LIN {X 0,Y 303.853,Z 837.936,A -85,B 0,C 180,E1 -16106.02,E2 -16106.02} C_VEL
LIN {X 0,Y 303.612,Z 839.547,A -85,B 0,C 180,E1 -16108.673,E2 -16108.673} C_VEL
LIN {X 0,Y 303.609,Z 839.78,A -85,B 0,C 180,E1 -16109.999,E2 -16109.999} C_VEL
LIN {X 0,Y 303.611,Z 839.586,A -85,B 0,C 180,E1 -16111.325,E2 -16111.325} C_VEL
LIN {X 0,Y 303.847,Z 838.029,A -85,B 0,C 180,E1 -16113.978,E2 -16113.978} C_VEL
LIN {X 0,Y 303.974,Z 836.663,A -85,B 0,C 180,E1 -16115.305,E2 -16115.305} C_VEL
LIN {X 0,Y 304.327,Z 833.787,A -85,B 0,C 180,E1 -16117.296,E2 -16117.296} C_VEL
LIN {X 0,Y 304.835,Z 829.878,A -85,B 0,C 180,E1 -16119.286,E2 -16119.286} C_VEL
LIN {X 0,Y 305.628,Z 824.814,A -85,B 0,C 180,E1 -16121.27,E2 -16121.27} C_VEL
LIN {X 0,Y 306.668,Z 818.43,A -85,B 0,C 180,E1 -16123.247,E2 -16123.247} C_VEL
LIN {X 0,Y 308.069,Z 810.481,A -85,B 0,C 180,E1 -16125.208,E2 -16125.208} C_VEL
LIN {X 0,Y 309.461,Z 802.349,A -85,B 0,C 180,E1 -16126.83,E2 -16126.83} C_VEL
LIN {X 0,Y 310.862,Z 792.359,A -85,B 0,C 180,E1 -16128.451,E2 -16128.451} C_VEL
LIN {X 0,Y 312.33,Z 781.127,A -85,B 0,C 180,E1 -16129.896,E2 -16129.896} C_VEL
LIN {X 0,Y 313.671,Z 770.081,A -85,B 0,C 180,E1 -16131.006,E2 -16131.006} C_VEL
LIN {X 0,Y 314.929,Z 757.587,A -85,B 0,C 180,E1 -16131.948,E2 -16131.948} C_VEL
LIN {X 0,Y 315.711,Z 745.352,A -85,B 0,C 180,E1 -16132.623,E2 -16132.623} C_VEL
LIN {X 0,Y 316.307,Z 733.163,A -85,B 0,C 180,E1 -16133.053,E2 -16133.053} C_VEL
LIN {X 0,Y 318.131,Z 657.232,A -85,B 0,C 180,E1 -16134.766,E2 -16134.766} C_VEL
LIN {X 0,Y 314.244,Z 634.232,A -85,B 0,C 180,E1 -16135.666,E2 -16135.666} C_VEL
LIN {X 0,Y 312.534,Z 625.542,A -85,B 0,C 180,E1 -16136.042,E2 -16136.042} C_VEL
LIN {X 0,Y 313.811,Z 610.673,A -85,B 0,C 180,E1 -16138.901,E2 -16138.901} C_VEL
LIN {X 0,Y 314.735,Z 599.426,A -85,B 0,C 180,E1 -16141.163,E2 -16141.163} C_VEL
LIN {X 0,Y 312.386,Z 587.67,A -85,B 0,C 180,E1 -16143.984,E2 -16143.984} C_VEL
LIN {X 0,Y 309.121,Z 574.667,A -85,B 0,C 180,E1 -16147.274,E2 -16147.274} C_VEL
LIN {X 0,Y 308.68,Z 573.104,A -85,B 0,C 180,E1 -16147.688,E2 -16147.688} C_VEL
LIN {X 0,Y 307.449,Z 571.218,A -85,B 0,C 180,E1 -16148.289,E2 -16148.289} C_VEL
LIN {X 0,Y 303.889,Z 568.949,A -85,B 0,C 180,E1 -16149.268,E2 -16149.268} C_VEL
LIN {X 0,Y 300.215,Z 566.767,A -85,B 0,C 180,E1 -16150.27,E2 -16150.27} C_VEL
LIN {X 0,Y 298.831,Z 564.916,A -85,B 0,C 180,E1 -16150.899,E2 -16150.899} C_VEL
LIN {X 0,Y 298.391,Z 563.319,A -85,B 0,C 180,E1 -16151.371,E2 -16151.371} C_VEL
LIN {X 0,Y 298.431,Z 563.292,A -85,B 0,C 180,E1 -16154.237,E2 -16154.237} C_VEL
LIN {X 0,Y 307.008,Z 587.38,A -85,B 0,C 180,E1 -16155.516,E2 -16155.516} C_VEL
LIN {X 0,Y 305.715,Z 636.753,A -85,B 0,C 180,E1 -16156.941,E2 -16156.941} C_VEL
LIN {X 0,Y 305.575,Z 650.861,A -85,B 0,C 180,E1 -16157.466,E2 -16157.466} C_VEL
LIN {X 0,Y 305.157,Z 664.019,A -85,B 0,C 180,E1 -16158.217,E2 -16158.217} C_VEL
LIN {X 0,Y 304.525,Z 676.406,A -85,B 0,C 180,E1 -16159.176,E2 -16159.176} C_VEL
LIN {X 0,Y 303.715,Z 689.144,A -85,B 0,C 180,E1 -16160.479,E2 -16160.479} C_VEL
LIN {X 0,Y 302.952,Z 699.146,A -85,B 0,C 180,E1 -16161.754,E2 -16161.754} C_VEL
LIN {X 0,Y 302.031,Z 709.642,A -85,B 0,C 180,E1 -16163.396,E2 -16163.396} C_VEL
LIN {X 0,Y 301.174,Z 718.74,A -85,B 0,C 180,E1 -16165.152,E2 -16165.152} C_VEL
LIN {X 0,Y 300.4,Z 726.936,A -85,B 0,C 180,E1 -16167.087,E2 -16167.087} C_VEL
LIN {X 0,Y 299.749,Z 733.339,A -85,B 0,C 180,E1 -16168.948,E2 -16168.948} C_VEL
LIN {X 0,Y 299.288,Z 739.52,A -85,B 0,C 180,E1 -16171.224,E2 -16171.224} C_VEL
LIN {X 0,Y 298.93,Z 744.17,A -85,B 0,C 180,E1 -16173.468,E2 -16173.468} C_VEL
LIN {X 0,Y 298.784,Z 746.542,A -85,B 0,C 180,E1 -16174.951,E2 -16174.951} C_VEL
LIN {X 0,Y 298.8,Z 748.429,A -85,B 0,C 180,E1 -16176.531,E2 -16176.531} C_VEL
LIN {X 0,Y 298.875,Z 749.634,A -85,B 0,C 180,E1 -16177.899,E2 -16177.899} C_VEL
LIN {X 0,Y 299.187,Z 750.596,A -85,B 0,C 180,E1 -16179.981,E2 -16179.981} C_VEL
LIN {X 0,Y 299.717,Z 750.5,A -85,B 0,C 180,E1 -16182.252,E2 -16182.252} C_VEL
LIN {X 0,Y 300.208,Z 749.793,A -85,B 0,C 180,E1 -16183.698,E2 -16183.698} C_VEL
LIN {X 0,Y 300.767,Z 748.669,A -85,B 0,C 180,E1 -16185.106,E2 -16185.106} C_VEL
LIN {X 0,Y 301.416,Z 747.031,A -85,B 0,C 180,E1 -16186.516,E2 -16186.516} C_VEL
LIN {X 0,Y 302.579,Z 743.644,A -85,B 0,C 180,E1 -16188.613,E2 -16188.613} C_VEL
LIN {X 0,Y 304.012,Z 739.036,A -85,B 0,C 180,E1 -16190.687,E2 -16190.687} C_VEL
LIN {X 0,Y 305.628,Z 733.047,A -85,B 0,C 180,E1 -16192.756,E2 -16192.756} C_VEL
LIN {X 0,Y 307.449,Z 725.584,A -85,B 0,C 180,E1 -16194.754,E2 -16194.754} C_VEL
LIN {X 0,Y 309.25,Z 717.437,A -85,B 0,C 180,E1 -16196.5,E2 -16196.5} C_VEL
LIN {X 0,Y 310.935,Z 708.306,A -85,B 0,C 180,E1 -16198.099,E2 -16198.099} C_VEL
LIN {X 0,Y 312.621,Z 698.14,A -85,B 0,C 180,E1 -16199.517,E2 -16199.517} C_VEL
LIN {X 0,Y 314.131,Z 686.583,A -85,B 0,C 180,E1 -16200.801,E2 -16200.801} C_VEL
LIN {X 0,Y 315.358,Z 674.542,A -85,B 0,C 180,E1 -16201.836,E2 -16201.836} C_VEL
LIN {X 0,Y 316.231,Z 660.72,A -85,B 0,C 180,E1 -16202.723,E2 -16202.723} C_VEL
LIN {X 0,Y 316.632,Z 647.103,A -85,B 0,C 180,E1 -16203.316,E2 -16203.316} C_VEL
LIN {X 0,Y 317.899,Z 617.446,A -85,B 0,C 180,E1 -16204.302,E2 -16204.302} C_VEL
LIN {X 0,Y 318.949,Z 597.845,A -85,B 0,C 180,E1 -16204.935,E2 -16204.935} C_VEL
LIN {X 0,Y 314.572,Z 589.417,A -85,B 0,C 180,E1 -16205.965,E2 -16205.965} C_VEL
LIN {X 0,Y 306.906,Z 576.235,A -85,B 0,C 180,E1 -16207.897,E2 -16207.897} C_VEL
LIN {X 0,Y 304.292,Z 572.293,A -85,B 0,C 180,E1 -16208.591,E2 -16208.591} C_VEL
LIN {X 0,Y 302.125,Z 569.115,A -85,B 0,C 180,E1 -16209.179,E2 -16209.179} C_VEL
LIN {X 0,Y 301.351,Z 567.986,A -85,B 0,C 180,E1 -16209.396,E2 -16209.396} C_VEL
LIN {X 0,Y 299.391,Z 565.714,A -85,B 0,C 180,E1 -16209.943,E2 -16209.943} C_VEL
LIN {X 0,Y 298.616,Z 563.282,A -85,B 0,C 180,E1 -16210.274,E2 -16210.274} C_VEL
LIN {X 0,Y 298.584,Z 563.287,A -85,B 0,C 180,E1 -16215.006,E2 -16215.006} C_VEL
LIN {X 0,Y 298.53,Z 563.298,A -85,B 0,C 180,E1 -16219.244,E2 -16219.244} C_VEL
LIN {X 0,Y 298.449,Z 563.309,A -85,B 0,C 180,E1 -16223.598,E2 -16223.598} C_VEL
LIN {X 0,Y 298.481,Z 563.304,A -85,B 0,C 180,E1 -16226.575,E2 -16226.575} C_VEL
LIN {X 0,Y 298.413,Z 563.313,A -85,B 0,C 180,E1 -16229.642,E2 -16229.642} C_VEL
LIN {X 0,Y 298.388,Z 563.317,A -85,B 0,C 180,E1 -16232.801,E2 -16232.801} C_VEL
LIN {X 0,Y 298.459,Z 563.304,A -85,B 0,C 180,E1 -16236.814,E2 -16236.814} C_VEL
LIN {X 0,Y 298.45,Z 563.309,A -85,B 0,C 180,E1 -16241.104,E2 -16241.104} C_VEL
LIN {X 0,Y 298.471,Z 563.304,A -85,B 0,C 180,E1 -16242.607,E2 -16242.607} C_VEL
LIN {X 0,Y 300.836,Z 570.374,A -85,B 0,C 180,E1 -16246.403,E2 -16246.403} C_VEL
LIN {X 0,Y 303.269,Z 578.289,A -85,B 0,C 180,E1 -16249.885,E2 -16249.885} C_VEL
LIN {X 0,Y 305.728,Z 587.467,A -85,B 0,C 180,E1 -16253.298,E2 -16253.298} C_VEL
LIN {X 0,Y 307.819,Z 597.274,A -85,B 0,C 180,E1 -16256.458,E2 -16256.458} C_VEL
LIN {X 0,Y 308.48,Z 601.915,A -85,B 0,C 180,E1 -16257.793,E2 -16257.793} C_VEL
LIN {X 0,Y 307.38,Z 607.823,A -85,B 0,C 180,E1 -16259.17,E2 -16259.17} C_VEL
LIN {X 0,Y 311.06,Z 628.758,A -85,B 0,C 180,E1 -16260.676,E2 -16260.676} C_VEL
LIN {X 0,Y 313.364,Z 646.451,A -85,B 0,C 180,E1 -16261.741,E2 -16261.741} C_VEL
LIN {X 0,Y 314.792,Z 663.123,A -85,B 0,C 180,E1 -16262.607,E2 -16262.607} C_VEL
LIN {X 0,Y 315.561,Z 682.154,A -85,B 0,C 180,E1 -16263.427,E2 -16263.427} C_VEL
LIN {X 0,Y 313.252,Z 724.371,A -85,B 0,C 180,E1 -16264.743,E2 -16264.743} C_VEL
LIN {X 0,Y 311.907,Z 737.532,A -85,B 0,C 180,E1 -16265.366,E2 -16265.366} C_VEL
LIN {X 0,Y 310.311,Z 749.164,A -85,B 0,C 180,E1 -16266.121,E2 -16266.121} C_VEL
LIN {X 0,Y 308.409,Z 760.554,A -85,B 0,C 180,E1 -16267.032,E2 -16267.032} C_VEL
LIN {X 0,Y 307.364,Z 773.902,A -85,B 0,C 180,E1 -16267.748,E2 -16267.748} C_VEL
LIN {X 0,Y 306.138,Z 785.541,A -85,B 0,C 180,E1 -16268.628,E2 -16268.628} C_VEL
LIN {X 0,Y 304.724,Z 796.825,A -85,B 0,C 180,E1 -16269.762,E2 -16269.762} C_VEL
LIN {X 0,Y 303.078,Z 808.262,A -85,B 0,C 180,E1 -16271.233,E2 -16271.233} C_VEL
LIN {X 0,Y 301.636,Z 817.897,A -85,B 0,C 180,E1 -16272.801,E2 -16272.801} C_VEL
LIN {X 0,Y 300.132,Z 827.345,A -85,B 0,C 180,E1 -16274.727,E2 -16274.727} C_VEL
LIN {X 0,Y 298.789,Z 835.261,A -85,B 0,C 180,E1 -16276.743,E2 -16276.743} C_VEL
LIN {X 0,Y 297.966,Z 840.605,A -85,B 0,C 180,E1 -16278.436,E2 -16278.436} C_VEL
LIN {X 0,Y 297.288,Z 845.825,A -85,B 0,C 180,E1 -16280.476,E2 -16280.476} C_VEL
LIN {X 0,Y 296.856,Z 849.862,A -85,B 0,C 180,E1 -16282.519,E2 -16282.519} C_VEL
LIN {X 0,Y 296.64,Z 852.837,A -85,B 0,C 180,E1 -16284.563,E2 -16284.563} C_VEL
LIN {X 0,Y 296.633,Z 854.265,A -85,B 0,C 180,E1 -16285.925,E2 -16285.925} C_VEL
LIN {X 0,Y 296.613,Z 855.272,A -85,B 0,C 180,E1 -16287.285,E2 -16287.285} C_VEL
LIN {X 0,Y 296.59,Z 855.887,A -85,B 0,C 180,E1 -16288.643,E2 -16288.643} C_VEL
LIN {X 0,Y 296.637,Z 856.105,A -85,B 0,C 180,E1 -16290.001,E2 -16290.001} C_VEL
LIN {X 0,Y 296.608,Z 855.258,A -85,B 0,C 180,E1 -16292.717,E2 -16292.717} C_VEL
LIN {X 0,Y 296.625,Z 854.245,A -85,B 0,C 180,E1 -16294.077,E2 -16294.077} C_VEL
LIN {X 0,Y 296.667,Z 852.404,A -85,B 0,C 180,E1 -16295.745,E2 -16295.745} C_VEL
LIN {X 0,Y 296.984,Z 848.58,A -85,B 0,C 180,E1 -16298.164,E2 -16298.164} C_VEL
LIN {X 0,Y 297.462,Z 844.157,A -85,B 0,C 180,E1 -16300.208,E2 -16300.208} C_VEL
LIN {X 0,Y 298.393,Z 837.421,A -85,B 0,C 180,E1 -16302.585,E2 -16302.585} C_VEL
LIN {X 0,Y 299.642,Z 830.074,A -85,B 0,C 180,E1 -16304.605,E2 -16304.605} C_VEL
LIN {X 0,Y 301.09,Z 821.3,A -85,B 0,C 180,E1 -16306.539,E2 -16306.539} C_VEL
LIN {X 0,Y 302.472,Z 811.371,A -85,B 0,C 180,E1 -16308.282,E2 -16308.282} C_VEL
LIN {X 0,Y 304.14,Z 800.779,A -85,B 0,C 180,E1 -16309.753,E2 -16309.753} C_VEL
LIN {X 0,Y 305.54,Z 790.516,A -85,B 0,C 180,E1 -16310.888,E2 -16310.888} C_VEL
LIN {X 0,Y 306.863,Z 778.19,A -85,B 0,C 180,E1 -16311.939,E2 -16311.939} C_VEL
LIN {X 0,Y 308.027,Z 765.239,A -85,B 0,C 180,E1 -16312.735,E2 -16312.735} C_VEL
LIN {X 0,Y 308.875,Z 752.279,A -85,B 0,C 180,E1 -16313.244,E2 -16313.244} C_VEL
LIN {X 0,Y 310.541,Z 681.414,A -85,B 0,C 180,E1 -16314.888,E2 -16314.888} C_VEL
LIN {X 0,Y 307.31,Z 650.705,A -85,B 0,C 180,E1 -16315.941,E2 -16315.941} C_VEL
LIN {X 0,Y 305.214,Z 635.339,A -85,B 0,C 180,E1 -16316.537,E2 -16316.537} C_VEL
LIN {X 0,Y 303.765,Z 612.724,A -85,B 0,C 180,E1 -16318.456,E2 -16318.456} C_VEL
LIN {X 0,Y 303.073,Z 604.261,A -85,B 0,C 180,E1 -16319.143,E2 -16319.143} C_VEL
LIN {X 0,Y 304.618,Z 592.104,A -85,B 0,C 180,E1 -16322.05,E2 -16322.05} C_VEL
LIN {X 0,Y 302.355,Z 581.022,A -85,B 0,C 180,E1 -16324.963,E2 -16324.963} C_VEL
LIN {X 0,Y 299.36,Z 567.37,A -85,B 0,C 180,E1 -16328.733,E2 -16328.733} C_VEL
LIN {X 0,Y 298.435,Z 563.311,A -85,B 0,C 180,E1 -16329.921,E2 -16329.921} C_VEL
LIN {X 0,Y 298.401,Z 563.308,A -85,B 0,C 180,E1 -16333.104,E2 -16333.104} C_VEL
LIN {X 0,Y 298.405,Z 563.311,A -85,B 0,C 180,E1 -16336.921,E2 -16336.921} C_VEL
LIN {X 0,Y 298.401,Z 563.317,A -85,B 0,C 180,E1 -16341.008,E2 -16341.008} C_VEL
LIN {X 0,Y 298.42,Z 563.299,A -85,B 0,C 180,E1 -16343.93,E2 -16343.93} C_VEL
LIN {X 0,Y 298.397,Z 563.302,A -85,B 0,C 180,E1 -16347.984,E2 -16347.984} C_VEL
LIN {X 0,Y 298.465,Z 563.307,A -85,B 0,C 180,E1 -16351.904,E2 -16351.904} C_VEL
LIN {X 0,Y 298.485,Z 563.284,A -85,B 0,C 180,E1 -16354.924,E2 -16354.924} C_VEL
LIN {X 0,Y 298.441,Z 563.309,A -85,B 0,C 180,E1 -16359.315,E2 -16359.315} C_VEL
LIN {X 0,Y 298.539,Z 563.271,A -85,B 0,C 180,E1 -16362.179,E2 -16362.179} C_VEL
LIN {X 0,Y 298.595,Z 563.287,A -85,B 0,C 180,E1 -16364.995,E2 -16364.995} C_VEL
LIN {X 0,Y 298.593,Z 563.266,A -85,B 0,C 180,E1 -16369.147,E2 -16369.147} C_VEL
LIN {X 0,Y 298.743,Z 563.264,A -85,B 0,C 180,E1 -16371.886,E2 -16371.886} C_VEL
LIN {X 0,Y 298.659,Z 563.279,A -85,B 0,C 180,E1 -16374.599,E2 -16374.599} C_VEL
LIN {X 0,Y 298.923,Z 563.232,A -85,B 0,C 180,E1 -16378.653,E2 -16378.653} C_VEL
LIN {X 0,Y 298.925,Z 563.25,A -85,B 0,C 180,E1 -16381.347,E2 -16381.347} C_VEL
LIN {X 0,Y 298.794,Z 563.254,A -85,B 0,C 180,E1 -16386.754,E2 -16386.754} C_VEL
LIN {X 0,Y 298.682,Z 563.281,A -85,B 0,C 180,E1 -16389.48,E2 -16389.48} C_VEL
LIN {X 0,Y 298.553,Z 563.278,A -85,B 0,C 180,E1 -16393.615,E2 -16393.615} C_VEL
LIN {X 0,Y 298.551,Z 563.295,A -85,B 0,C 180,E1 -16396.409,E2 -16396.409} C_VEL
LIN {X 0,Y 298.513,Z 563.28,A -85,B 0,C 180,E1 -16399.654,E2 -16399.654} C_VEL
LIN {X 0,Y 298.46,Z 563.303,A -85,B 0,C 180,E1 -16403.598,E2 -16403.598} C_VEL
LIN {X 0,Y 298.487,Z 563.294,A -85,B 0,C 180,E1 -16406.575,E2 -16406.575} C_VEL
LIN {X 0,Y 298.419,Z 563.305,A -85,B 0,C 180,E1 -16409.641,E2 -16409.641} C_VEL
LIN {X 0,Y 298.397,Z 563.318,A -85,B 0,C 180,E1 -16412.8,E2 -16412.8} C_VEL
LIN {X 0,Y 298.466,Z 563.307,A -85,B 0,C 180,E1 -16416.812,E2 -16416.812} C_VEL
LIN {X 0,Y 298.39,Z 563.319,A -85,B 0,C 180,E1 -16421.088,E2 -16421.088} C_VEL
LIN {X 0,Y 298.401,Z 563.307,A -85,B 0,C 180,E1 -16423.103,E2 -16423.103} C_VEL
LIN {X 0,Y 298.406,Z 563.29,A -85,B 0,C 180,E1 -16426.921,E2 -16426.921} C_VEL
LIN {X 0,Y 298.43,Z 563.37,A -85,B 0,C 180,E1 -16430.401,E2 -16430.401} C_VEL
LIN {X 0,Y 302.152,Z 575.058,A -85,B 0,C 180,E1 -16433.365,E2 -16433.365} C_VEL
LIN {X 0,Y 305.463,Z 587.296,A -85,B 0,C 180,E1 -16436.257,E2 -16436.257} C_VEL
LIN {X 0,Y 308.042,Z 598.396,A -85,B 0,C 180,E1 -16438.732,E2 -16438.732} C_VEL
LIN {X 0,Y 308.779,Z 602.347,A -85,B 0,C 180,E1 -16439.574,E2 -16439.574} C_VEL
LIN {X 0,Y 307.17,Z 620.347,A -85,B 0,C 180,E1 -16442.767,E2 -16442.767} C_VEL
LIN {X 0,Y 306.845,Z 624.941,A -85,B 0,C 180,E1 -16443.537,E2 -16443.537} C_VEL
LIN {X 0,Y 311.493,Z 653.75,A -85,B 0,C 180,E1 -16444.695,E2 -16444.695} C_VEL
LIN {X 0,Y 311.626,Z 659.554,A -85,B 0,C 180,E1 -16444.852,E2 -16444.852} C_VEL
LIN {X 0,Y 309.66,Z 736.424,A -85,B 0,C 180,E1 -16446.642,E2 -16446.642} C_VEL
LIN {X 0,Y 308.963,Z 749.181,A -85,B 0,C 180,E1 -16447.162,E2 -16447.162} C_VEL
LIN {X 0,Y 307.876,Z 762.003,A -85,B 0,C 180,E1 -16447.961,E2 -16447.961} C_VEL
LIN {X 0,Y 306.553,Z 774.243,A -85,B 0,C 180,E1 -16449.008,E2 -16449.008} C_VEL
LIN {X 0,Y 305.168,Z 784.527,A -85,B 0,C 180,E1 -16450.141,E2 -16450.141} C_VEL
LIN {X 0,Y 303.816,Z 794.443,A -85,B 0,C 180,E1 -16451.52,E2 -16451.52} C_VEL
LIN {X 0,Y 302.426,Z 803.706,A -85,B 0,C 180,E1 -16453.112,E2 -16453.112} C_VEL
LIN {X 0,Y 300.731,Z 813.082,A -85,B 0,C 180,E1 -16455.103,E2 -16455.103} C_VEL
LIN {X 0,Y 299.443,Z 820.531,A -85,B 0,C 180,E1 -16457.116,E2 -16457.116} C_VEL
LIN {X 0,Y 298.397,Z 826.513,A -85,B 0,C 180,E1 -16459.138,E2 -16459.138} C_VEL
LIN {X 0,Y 297.631,Z 831.239,A -85,B 0,C 180,E1 -16461.17,E2 -16461.17} C_VEL
LIN {X 0,Y 297.107,Z 835.247,A -85,B 0,C 180,E1 -16463.467,E2 -16463.467} C_VEL
LIN {X 0,Y 296.769,Z 838.129,A -85,B 0,C 180,E1 -16465.925,E2 -16465.925} C_VEL
LIN {X 0,Y 296.531,Z 839.74,A -85,B 0,C 180,E1 -16468.641,E2 -16468.641} C_VEL
LIN {X 0,Y 296.525,Z 839.973,A -85,B 0,C 180,E1 -16469.999,E2 -16469.999} C_VEL
LIN {X 0,Y 296.53,Z 839.779,A -85,B 0,C 180,E1 -16471.357,E2 -16471.357} C_VEL
LIN {X 0,Y 296.764,Z 838.222,A -85,B 0,C 180,E1 -16474.073,E2 -16474.073} C_VEL
LIN {X 0,Y 297.076,Z 835.498,A -85,B 0,C 180,E1 -16476.48,E2 -16476.48} C_VEL
LIN {X 0,Y 297.606,Z 831.47,A -85,B 0,C 180,E1 -16478.828,E2 -16478.828} C_VEL
LIN {X 0,Y 298.362,Z 826.807,A -85,B 0,C 180,E1 -16480.861,E2 -16480.861} C_VEL
LIN {X 0,Y 299.394,Z 820.897,A -85,B 0,C 180,E1 -16482.884,E2 -16482.884} C_VEL
LIN {X 0,Y 300.668,Z 813.536,A -85,B 0,C 180,E1 -16484.898,E2 -16484.898} C_VEL
LIN {X 0,Y 302.078,Z 805.993,A -85,B 0,C 180,E1 -16486.558,E2 -16486.558} C_VEL
LIN {X 0,Y 303.654,Z 795.708,A -85,B 0,C 180,E1 -16488.388,E2 -16488.388} C_VEL
LIN {X 0,Y 305.131,Z 785.367,A -85,B 0,C 180,E1 -16489.859,E2 -16489.859} C_VEL
LIN {X 0,Y 306.481,Z 775.33,A -85,B 0,C 180,E1 -16490.994,E2 -16490.994} C_VEL
LIN {X 0,Y 307.813,Z 763.399,A -85,B 0,C 180,E1 -16492.041,E2 -16492.041} C_VEL
LIN {X 0,Y 308.86,Z 750.384,A -85,B 0,C 180,E1 -16492.888,E2 -16492.888} C_VEL
LIN {X 0,Y 309.637,Z 737.22,A -85,B 0,C 180,E1 -16493.446,E2 -16493.446} C_VEL
LIN {X 0,Y 311.73,Z 659.363,A -85,B 0,C 180,E1 -16495.257,E2 -16495.257} C_VEL
LIN {X 0,Y 309.107,Z 642.217,A -85,B 0,C 180,E1 -16495.923,E2 -16495.923} C_VEL
LIN {X 0,Y 305.998,Z 625.586,A -85,B 0,C 180,E1 -16496.668,E2 -16496.668} C_VEL
LIN {X 0,Y 307.473,Z 608.89,A -85,B 0,C 180,E1 -16499.915,E2 -16499.915} C_VEL
LIN {X 0,Y 308.081,Z 602.29,A -85,B 0,C 180,E1 -16501.262,E2 -16501.262} C_VEL
LIN {X 0,Y 306.536,Z 593.373,A -85,B 0,C 180,E1 -16503.382,E2 -16503.382} C_VEL
LIN {X 0,Y 303.751,Z 581.527,A -85,B 0,C 180,E1 -16506.401,E2 -16506.401} C_VEL
LIN {X 0,Y 300.486,Z 569.988,A -85,B 0,C 180,E1 -16509.481,E2 -16509.481} C_VEL
LIN {X 0,Y 298.831,Z 564.916,A -85,B 0,C 180,E1 -16510.899,E2 -16510.899} C_VEL
LIN {X 0,Y 298.207,Z 564.181,A -85,B 0,C 180,E1 -16511.434,E2 -16511.434} C_VEL
LIN {X 0,Y 297.663,Z 564.724,A -85,B 0,C 180,E1 -16512.005,E2 -16512.005} C_VEL
LIN {X 0,Y 297.105,Z 566.972,A -85,B 0,C 180,E1 -16512.788,E2 -16512.788} C_VEL
LIN {X 0,Y 296.868,Z 571.244,A -85,B 0,C 180,E1 -16513.605,E2 -16513.605} C_VEL
LIN {X 0,Y 297.126,Z 576.758,A -85,B 0,C 180,E1 -16514.323,E2 -16514.323} C_VEL
LIN {X 0,Y 298.201,Z 582.694,A -85,B 0,C 180,E1 -16514.845,E2 -16514.845} C_VEL
LIN {X 0,Y 298.815,Z 584.718,A -85,B 0,C 180,E1 -16514.965,E2 -16514.965} C_VEL
LIN {X 0,Y 300.204,Z 588.9,A -85,B 0,C 180,E1 -16515.177,E2 -16515.177} C_VEL
LIN {X 0,Y 298.863,Z 635.716,A -85,B 0,C 180,E1 -16516.565,E2 -16516.565} C_VEL
LIN {X 0,Y 298.706,Z 650.873,A -85,B 0,C 180,E1 -16517.119,E2 -16517.119} C_VEL
LIN {X 0,Y 298.267,Z 664.834,A -85,B 0,C 180,E1 -16517.928,E2 -16517.928} C_VEL
LIN {X 0,Y 297.61,Z 677.799,A -85,B 0,C 180,E1 -16518.963,E2 -16518.963} C_VEL
LIN {X 0,Y 296.761,Z 690.075,A -85,B 0,C 180,E1 -16520.251,E2 -16520.251} C_VEL
LIN {X 0,Y 295.961,Z 700.332,A -85,B 0,C 180,E1 -16521.591,E2 -16521.591} C_VEL
LIN {X 0,Y 295.03,Z 710.591,A -85,B 0,C 180,E1 -16523.236,E2 -16523.236} C_VEL
LIN {X 0,Y 294.147,Z 719.592,A -85,B 0,C 180,E1 -16525.01,E2 -16525.01} C_VEL
LIN {X 0,Y 293.374,Z 727.748,A -85,B 0,C 180,E1 -16526.973,E2 -16526.973} C_VEL
LIN {X 0,Y 292.711,Z 734.342,A -85,B 0,C 180,E1 -16528.921,E2 -16528.921} C_VEL
LIN {X 0,Y 292.228,Z 740.543,A -85,B 0,C 180,E1 -16531.249,E2 -16531.249} C_VEL
LIN {X 0,Y 291.873,Z 745.38,A -85,B 0,C 180,E1 -16533.637,E2 -16533.637} C_VEL
LIN {X 0,Y 291.752,Z 748.574,A -85,B 0,C 180,E1 -16535.826,E2 -16535.826} C_VEL
LIN {X 0,Y 291.792,Z 750.114,A -85,B 0,C 180,E1 -16537.333,E2 -16537.333} C_VEL
LIN {X 0,Y 292.13,Z 751.538,A -85,B 0,C 180,E1 -16539.754,E2 -16539.754} C_VEL
LIN {X 0,Y 292.577,Z 751.747,A -85,B 0,C 180,E1 -16541.804,E2 -16541.804} C_VEL
LIN {X 0,Y 293.142,Z 751.226,A -85,B 0,C 180,E1 -16543.527,E2 -16543.527} C_VEL
LIN {X 0,Y 293.624,Z 750.434,A -85,B 0,C 180,E1 -16544.735,E2 -16544.735} C_VEL
LIN {X 0,Y 294.293,Z 749.041,A -85,B 0,C 180,E1 -16546.184,E2 -16546.184} C_VEL
LIN {X 0,Y 295.446,Z 746.059,A -85,B 0,C 180,E1 -16548.334,E2 -16548.334} C_VEL
LIN {X 0,Y 296.901,Z 741.881,A -85,B 0,C 180,E1 -16550.462,E2 -16550.462} C_VEL
LIN {X 0,Y 298.724,Z 735.75,A -85,B 0,C 180,E1 -16552.788,E2 -16552.788} C_VEL
LIN {X 0,Y 300.746,Z 728.221,A -85,B 0,C 180,E1 -16554.973,E2 -16554.973} C_VEL
LIN {X 0,Y 302.671,Z 720.291,A -85,B 0,C 180,E1 -16556.779,E2 -16556.779} C_VEL
LIN {X 0,Y 304.542,Z 710.854,A -85,B 0,C 180,E1 -16558.513,E2 -16558.513} C_VEL
LIN {X 0,Y 306.389,Z 700.702,A -85,B 0,C 180,E1 -16560,E2 -16560} C_VEL
LIN {X 0,Y 307.999,Z 689.593,A -85,B 0,C 180,E1 -16561.307,E2 -16561.307} C_VEL
LIN {X 0,Y 309.333,Z 677.861,A -85,B 0,C 180,E1 -16562.389,E2 -16562.389} C_VEL
LIN {X 0,Y 310.328,Z 664.967,A -85,B 0,C 180,E1 -16563.286,E2 -16563.286} C_VEL
LIN {X 0,Y 310.847,Z 652.053,A -85,B 0,C 180,E1 -16563.921,E2 -16563.921} C_VEL
LIN {X 0,Y 311.957,Z 624.36,A -85,B 0,C 180,E1 -16564.889,E2 -16564.889} C_VEL
LIN {X 0,Y 313.475,Z 600.699,A -85,B 0,C 180,E1 -16565.657,E2 -16565.657} C_VEL
LIN {X 0,Y 309.983,Z 593.909,A -85,B 0,C 180,E1 -16566.53,E2 -16566.53} C_VEL
LIN {X 0,Y 302.781,Z 581.278,A -85,B 0,C 180,E1 -16568.447,E2 -16568.447} C_VEL
LIN {X 0,Y 299.761,Z 576.856,A -85,B 0,C 180,E1 -16569.273,E2 -16569.273} C_VEL
LIN {X 0,Y 297.51,Z 573.44,A -85,B 0,C 180,E1 -16569.947,E2 -16569.947} C_VEL
LIN {X 0,Y 295.318,Z 570.414,A -85,B 0,C 180,E1 -16570.607,E2 -16570.607} C_VEL
LIN {X 0,Y 294.654,Z 569.199,A -85,B 0,C 180,E1 -16570.826,E2 -16570.826} C_VEL
LIN {X 0,Y 292.355,Z 566.759,A -85,B 0,C 180,E1 -16571.522,E2 -16571.522} C_VEL
LIN {X 0,Y 291.502,Z 564.171,A -85,B 0,C 180,E1 -16571.949,E2 -16571.949} C_VEL
LIN {X 0,Y 291.546,Z 564.161,A -85,B 0,C 180,E1 -16575.377,E2 -16575.377} C_VEL
LIN {X 0,Y 291.442,Z 564.181,A -85,B 0,C 180,E1 -16579.875,E2 -16579.875} C_VEL
LIN {X 0,Y 291.392,Z 564.187,A -85,B 0,C 180,E1 -16584.206,E2 -16584.206} C_VEL
LIN {X 0,Y 291.414,Z 564.184,A -85,B 0,C 180,E1 -16587.272,E2 -16587.272} C_VEL
LIN {X 0,Y 291.329,Z 564.196,A -85,B 0,C 180,E1 -16590.438,E2 -16590.438} C_VEL
LIN {X 0,Y 291.337,Z 564.192,A -85,B 0,C 180,E1 -16593.699,E2 -16593.699} C_VEL
LIN {X 0,Y 291.395,Z 564.181,A -85,B 0,C 180,E1 -16597.262,E2 -16597.262} C_VEL
LIN {X 0,Y 291.4,Z 564.248,A -85,B 0,C 180,E1 -16600.631,E2 -16600.631} C_VEL
LIN {X 0,Y 293.267,Z 569.628,A -85,B 0,C 180,E1 -16604.036,E2 -16604.036} C_VEL
LIN {X 0,Y 294.901,Z 574.551,A -85,B 0,C 180,E1 -16606.624,E2 -16606.624} C_VEL
LIN {X 0,Y 297.122,Z 581.906,A -85,B 0,C 180,E1 -16609.895,E2 -16609.895} C_VEL
LIN {X 0,Y 299.22,Z 590.028,A -85,B 0,C 180,E1 -16612.995,E2 -16612.995} C_VEL
LIN {X 0,Y 301.082,Z 598.793,A -85,B 0,C 180,E1 -16615.931,E2 -16615.931} C_VEL
LIN {X 0,Y 301.811,Z 603.371,A -85,B 0,C 180,E1 -16617.338,E2 -16617.338} C_VEL
LIN {X 0,Y 301.456,Z 605.988,A -85,B 0,C 180,E1 -16618.007,E2 -16618.007} C_VEL
LIN {X 0,Y 305.162,Z 627.035,A -85,B 0,C 180,E1 -16619.639,E2 -16619.639} C_VEL
LIN {X 0,Y 307.55,Z 645.152,A -85,B 0,C 180,E1 -16620.811,E2 -16620.811} C_VEL
LIN {X 0,Y 309.122,Z 663.349,A -85,B 0,C 180,E1 -16621.801,E2 -16621.801} C_VEL
LIN {X 0,Y 309.771,Z 682.896,A -85,B 0,C 180,E1 -16622.686,E2 -16622.686} C_VEL
LIN {X 0,Y 307.431,Z 723.239,A -85,B 0,C 180,E1 -16623.98,E2 -16623.98} C_VEL
LIN {X 0,Y 305.891,Z 737.363,A -85,B 0,C 180,E1 -16624.666,E2 -16624.666} C_VEL
LIN {X 0,Y 303.891,Z 750.637,A -85,B 0,C 180,E1 -16625.584,E2 -16625.584} C_VEL
LIN {X 0,Y 301.79,Z 762.196,A -85,B 0,C 180,E1 -16626.589,E2 -16626.589} C_VEL
LIN {X 0,Y 300.672,Z 774.996,A -85,B 0,C 180,E1 -16627.316,E2 -16627.316} C_VEL
LIN {X 0,Y 299.328,Z 787.124,A -85,B 0,C 180,E1 -16628.298,E2 -16628.298} C_VEL
LIN {X 0,Y 297.858,Z 798.06,A -85,B 0,C 180,E1 -16629.454,E2 -16629.454} C_VEL
LIN {X 0,Y 296.166,Z 809.207,A -85,B 0,C 180,E1 -16630.958,E2 -16630.958} C_VEL
LIN {X 0,Y 294.712,Z 818.444,A -85,B 0,C 180,E1 -16632.532,E2 -16632.532} C_VEL
LIN {X 0,Y 293.225,Z 827.157,A -85,B 0,C 180,E1 -16634.359,E2 -16634.359} C_VEL
LIN {X 0,Y 291.864,Z 835.072,A -85,B 0,C 180,E1 -16636.423,E2 -16636.423} C_VEL
LIN {X 0,Y 290.976,Z 840.414,A -85,B 0,C 180,E1 -16638.154,E2 -16638.154} C_VEL
LIN {X 0,Y 290.266,Z 845.634,A -85,B 0,C 180,E1 -16640.243,E2 -16640.243} C_VEL
LIN {X 0,Y 289.807,Z 849.671,A -85,B 0,C 180,E1 -16642.336,E2 -16642.336} C_VEL
LIN {X 0,Y 289.556,Z 852.644,A -85,B 0,C 180,E1 -16644.43,E2 -16644.43} C_VEL
LIN {X 0,Y 289.53,Z 854.072,A -85,B 0,C 180,E1 -16645.825,E2 -16645.825} C_VEL
LIN {X 0,Y 289.538,Z 855.08,A -85,B 0,C 180,E1 -16647.219,E2 -16647.219} C_VEL
LIN {X 0,Y 289.507,Z 855.694,A -85,B 0,C 180,E1 -16648.61,E2 -16648.61} C_VEL
LIN {X 0,Y 289.549,Z 855.913,A -85,B 0,C 180,E1 -16650.001,E2 -16650.001} C_VEL
LIN {X 0,Y 289.533,Z 855.066,A -85,B 0,C 180,E1 -16652.784,E2 -16652.784} C_VEL
LIN {X 0,Y 289.523,Z 854.052,A -85,B 0,C 180,E1 -16654.177,E2 -16654.177} C_VEL
LIN {X 0,Y 289.558,Z 852.505,A -85,B 0,C 180,E1 -16655.656,E2 -16655.656} C_VEL
LIN {X 0,Y 289.922,Z 848.386,A -85,B 0,C 180,E1 -16658.364,E2 -16658.364} C_VEL
LIN {X 0,Y 290.454,Z 843.964,A -85,B 0,C 180,E1 -16660.457,E2 -16660.457} C_VEL
LIN {X 0,Y 291.412,Z 837.227,A -85,B 0,C 180,E1 -16662.891,E2 -16662.891} C_VEL
LIN {X 0,Y 292.748,Z 829.882,A -85,B 0,C 180,E1 -16664.957,E2 -16664.957} C_VEL
LIN {X 0,Y 294.02,Z 822.387,A -85,B 0,C 180,E1 -16666.67,E2 -16666.67} C_VEL
LIN {X 0,Y 295.386,Z 813.287,A -85,B 0,C 180,E1 -16668.377,E2 -16668.377} C_VEL
LIN {X 0,Y 297.029,Z 803.153,A -85,B 0,C 180,E1 -16669.885,E2 -16669.885} C_VEL
LIN {X 0,Y 298.683,Z 791.905,A -85,B 0,C 180,E1 -16671.21,E2 -16671.21} C_VEL
LIN {X 0,Y 300.058,Z 780.212,A -85,B 0,C 180,E1 -16672.282,E2 -16672.282} C_VEL
LIN {X 0,Y 301.321,Z 767.308,A -85,B 0,C 180,E1 -16673.134,E2 -16673.134} C_VEL
LIN {X 0,Y 302.271,Z 754.649,A -85,B 0,C 180,E1 -16673.692,E2 -16673.692} C_VEL
LIN {X 0,Y 303.027,Z 729.922,A -85,B 0,C 180,E1 -16674.311,E2 -16674.311} C_VEL
LIN {X 0,Y 304.059,Z 681.164,A -85,B 0,C 180,E1 -16675.46,E2 -16675.46} C_VEL
LIN {X 0,Y 300.917,Z 651.415,A -85,B 0,C 180,E1 -16676.514,E2 -16676.514} C_VEL
LIN {X 0,Y 298.692,Z 635.206,A -85,B 0,C 180,E1 -16677.161,E2 -16677.161} C_VEL
LIN {X 0,Y 297.434,Z 613.946,A -85,B 0,C 180,E1 -16679.042,E2 -16679.042} C_VEL
LIN {X 0,Y 296.535,Z 601.421,A -85,B 0,C 180,E1 -16680.143,E2 -16680.143} C_VEL
LIN {X 0,Y 297.592,Z 592.905,A -85,B 0,C 180,E1 -16682.235,E2 -16682.235} C_VEL
LIN {X 0,Y 294.791,Z 579.626,A -85,B 0,C 180,E1 -16685.847,E2 -16685.847} C_VEL
LIN {X 0,Y 291.861,Z 566.445,A -85,B 0,C 180,E1 -16689.596,E2 -16689.596} C_VEL
LIN {X 0,Y 291.386,Z 564.19,A -85,B 0,C 180,E1 -16690.322,E2 -16690.322} C_VEL
LIN {X 0,Y 291.316,Z 564.185,A -85,B 0,C 180,E1 -16694.398,E2 -16694.398} C_VEL
LIN {X 0,Y 291.329,Z 564.181,A -85,B 0,C 180,E1 -16698.404,E2 -16698.404} C_VEL
LIN {X 0,Y 291.35,Z 564.193,A -85,B 0,C 180,E1 -16701.158,E2 -16701.158} C_VEL
LIN {X 0,Y 291.363,Z 564.183,A -85,B 0,C 180,E1 -16704.626,E2 -16704.626} C_VEL
LIN {X 0,Y 291.374,Z 564.177,A -85,B 0,C 180,E1 -16707.951,E2 -16707.951} C_VEL
LIN {X 0,Y 291.384,Z 564.185,A -85,B 0,C 180,E1 -16711.159,E2 -16711.159} C_VEL
LIN {X 0,Y 291.417,Z 564.169,A -85,B 0,C 180,E1 -16714.272,E2 -16714.272} C_VEL
LIN {X 0,Y 291.376,Z 564.182,A -85,B 0,C 180,E1 -16717.299,E2 -16717.299} C_VEL
LIN {X 0,Y 291.46,Z 564.172,A -85,B 0,C 180,E1 -16720.27,E2 -16720.27} C_VEL
LIN {X 0,Y 291.542,Z 564.164,A -85,B 0,C 180,E1 -16724.635,E2 -16724.635} C_VEL
LIN {X 0,Y 291.537,Z 564.146,A -85,B 0,C 180,E1 -16728.881,E2 -16728.881} C_VEL
LIN {X 0,Y 291.689,Z 564.14,A -85,B 0,C 180,E1 -16731.688,E2 -16731.688} C_VEL
LIN {X 0,Y 291.629,Z 564.155,A -85,B 0,C 180,E1 -16734.468,E2 -16734.468} C_VEL
LIN {X 0,Y 291.889,Z 564.107,A -85,B 0,C 180,E1 -16738.62,E2 -16738.62} C_VEL
LIN {X 0,Y 291.891,Z 564.127,A -85,B 0,C 180,E1 -16741.38,E2 -16741.38} C_VEL
LIN {X 0,Y 291.743,Z 564.135,A -85,B 0,C 180,E1 -16746.918,E2 -16746.918} C_VEL
LIN {X 0,Y 291.631,Z 564.156,A -85,B 0,C 180,E1 -16749.712,E2 -16749.712} C_VEL
LIN {X 0,Y 291.523,Z 564.156,A -85,B 0,C 180,E1 -16753.95,E2 -16753.95} C_VEL
LIN {X 0,Y 291.489,Z 564.173,A -85,B 0,C 180,E1 -16756.818,E2 -16756.818} C_VEL
LIN {X 0,Y 291.453,Z 564.16,A -85,B 0,C 180,E1 -16759.875,E2 -16759.875} C_VEL
LIN {X 0,Y 291.401,Z 564.174,A -85,B 0,C 180,E1 -16764.205,E2 -16764.205} C_VEL
LIN {X 0,Y 291.421,Z 564.181,A -85,B 0,C 180,E1 -16767.272,E2 -16767.272} C_VEL
LIN {X 0,Y 291.336,Z 564.181,A -85,B 0,C 180,E1 -16770.437,E2 -16770.437} C_VEL
LIN {X 0,Y 291.347,Z 564.197,A -85,B 0,C 180,E1 -16773.698,E2 -16773.698} C_VEL
LIN {X 0,Y 291.396,Z 564.19,A -85,B 0,C 180,E1 -16777.258,E2 -16777.258} C_VEL
LIN {X 0,Y 291.337,Z 564.193,A -85,B 0,C 180,E1 -16780.642,E2 -16780.642} C_VEL
LIN {X 0,Y 291.293,Z 564.2,A -85,B 0,C 180,E1 -16784.402,E2 -16784.402} C_VEL
LIN {X 0,Y 291.329,Z 564.174,A -85,B 0,C 180,E1 -16788.404,E2 -16788.404} C_VEL
LIN {X 0,Y 291.389,Z 564.228,A -85,B 0,C 180,E1 -16789.557,E2 -16789.557} C_VEL
LIN {X 0,Y 295.468,Z 576.807,A -85,B 0,C 180,E1 -16792.812,E2 -16792.812} C_VEL
LIN {X 0,Y 298.584,Z 588.234,A -85,B 0,C 180,E1 -16795.603,E2 -16795.603} C_VEL
LIN {X 0,Y 301.396,Z 600.311,A -85,B 0,C 180,E1 -16798.354,E2 -16798.354} C_VEL
LIN {X 0,Y 302.153,Z 605.135,A -85,B 0,C 180,E1 -16799.386,E2 -16799.386} C_VEL
LIN {X 0,Y 300.391,Z 624.096,A -85,B 0,C 180,E1 -16802.755,E2 -16802.755} C_VEL
LIN {X 0,Y 300.353,Z 625.317,A -85,B 0,C 180,E1 -16802.932,E2 -16802.932} C_VEL
LIN {X 0,Y 304.632,Z 651.72,A -85,B 0,C 180,E1 -16804.028,E2 -16804.028} C_VEL
LIN {X 0,Y 305.272,Z 657.467,A -85,B 0,C 180,E1 -16804.235,E2 -16804.235} C_VEL
LIN {X 0,Y 303.171,Z 736.554,A -85,B 0,C 180,E1 -16806.111,E2 -16806.111} C_VEL
LIN {X 0,Y 302.451,Z 749.34,A -85,B 0,C 180,E1 -16806.641,E2 -16806.641} C_VEL
LIN {X 0,Y 301.487,Z 761.103,A -85,B 0,C 180,E1 -16807.378,E2 -16807.378} C_VEL
LIN {X 0,Y 300.358,Z 771.034,A -85,B 0,C 180,E1 -16808.194,E2 -16808.194} C_VEL
LIN {X 0,Y 298.894,Z 781.961,A -85,B 0,C 180,E1 -16809.347,E2 -16809.347} C_VEL
LIN {X 0,Y 297.465,Z 791.987,A -85,B 0,C 180,E1 -16810.684,E2 -16810.684} C_VEL
LIN {X 0,Y 295.963,Z 802.149,A -85,B 0,C 180,E1 -16812.375,E2 -16812.375} C_VEL
LIN {X 0,Y 294.454,Z 810.38,A -85,B 0,C 180,E1 -16814.068,E2 -16814.068} C_VEL
LIN {X 0,Y 292.912,Z 818.406,A -85,B 0,C 180,E1 -16816.116,E2 -16816.116} C_VEL
LIN {X 0,Y 291.742,Z 824.868,A -85,B 0,C 180,E1 -16818.183,E2 -16818.183} C_VEL
LIN {X 0,Y 290.844,Z 830.005,A -85,B 0,C 180,E1 -16820.261,E2 -16820.261} C_VEL
LIN {X 0,Y 290.248,Z 833.976,A -85,B 0,C 180,E1 -16822.346,E2 -16822.346} C_VEL
LIN {X 0,Y 289.83,Z 836.904,A -85,B 0,C 180,E1 -16824.433,E2 -16824.433} C_VEL
LIN {X 0,Y 289.689,Z 838.323,A -85,B 0,C 180,E1 -16825.825,E2 -16825.825} C_VEL
LIN {X 0,Y 289.453,Z 839.932,A -85,B 0,C 180,E1 -16828.608,E2 -16828.608} C_VEL
LIN {X 0,Y 289.442,Z 840.165,A -85,B 0,C 180,E1 -16829.999,E2 -16829.999} C_VEL
LIN {X 0,Y 289.451,Z 839.971,A -85,B 0,C 180,E1 -16831.39,E2 -16831.39} C_VEL
LIN {X 0,Y 289.685,Z 838.414,A -85,B 0,C 180,E1 -16834.173,E2 -16834.173} C_VEL
LIN {X 0,Y 289.995,Z 835.916,A -85,B 0,C 180,E1 -16836.468,E2 -16836.468} C_VEL
LIN {X 0,Y 290.382,Z 832.964,A -85,B 0,C 180,E1 -16838.348,E2 -16838.348} C_VEL
LIN {X 0,Y 291.091,Z 828.686,A -85,B 0,C 180,E1 -16840.431,E2 -16840.431} C_VEL
LIN {X 0,Y 292.055,Z 823.224,A -85,B 0,C 180,E1 -16842.507,E2 -16842.507} C_VEL
LIN {X 0,Y 293.317,Z 816.367,A -85,B 0,C 180,E1 -16844.57,E2 -16844.57} C_VEL
LIN {X 0,Y 294.98,Z 807.771,A -85,B 0,C 180,E1 -16846.611,E2 -16846.611} C_VEL
LIN {X 0,Y 296.521,Z 798.769,A -85,B 0,C 180,E1 -16848.339,E2 -16848.339} C_VEL
LIN {X 0,Y 298.066,Z 788.041,A -85,B 0,C 180,E1 -16849.991,E2 -16849.991} C_VEL
LIN {X 0,Y 299.673,Z 777.034,A -85,B 0,C 180,E1 -16851.314,E2 -16851.314} C_VEL
LIN {X 0,Y 300.933,Z 766.624,A -85,B 0,C 180,E1 -16852.301,E2 -16852.301} C_VEL
LIN {X 0,Y 302.091,Z 754.082,A -85,B 0,C 180,E1 -16853.205,E2 -16853.205} C_VEL
LIN {X 0,Y 302.976,Z 740.752,A -85,B 0,C 180,E1 -16853.858,E2 -16853.858} C_VEL
LIN {X 0,Y 303.538,Z 724.676,A -85,B 0,C 180,E1 -16854.31,E2 -16854.31} C_VEL
LIN {X 0,Y 305.239,Z 658.779,A -85,B 0,C 180,E1 -16855.85,E2 -16855.85} C_VEL
LIN {X 0,Y 301.005,Z 633.913,A -85,B 0,C 180,E1 -16856.895,E2 -16856.895} C_VEL
LIN {X 0,Y 299.445,Z 625.772,A -85,B 0,C 180,E1 -16857.278,E2 -16857.278} C_VEL
LIN {X 0,Y 301.021,Z 608.81,A -85,B 0,C 180,E1 -16860.641,E2 -16860.641} C_VEL
LIN {X 0,Y 301.455,Z 603.988,A -85,B 0,C 180,E1 -16861.636,E2 -16861.636} C_VEL
LIN {X 0,Y 299.837,Z 595.02,A -85,B 0,C 180,E1 -16863.825,E2 -16863.825} C_VEL
LIN {X 0,Y 296.97,Z 582.787,A -85,B 0,C 180,E1 -16866.992,E2 -16866.992} C_VEL
LIN {X 0,Y 293.353,Z 570.687,A -85,B 0,C 180,E1 -16870.302,E2 -16870.302} C_VEL
LIN {X 0,Y 291.36,Z 564.179,A -85,B 0,C 180,E1 -16872.234,E2 -16872.234} C_VEL
LIN {X 0,Y 291.409,Z 564.367,A -85,B 0,C 180,E1 -16873.86,E2 -16873.86} C_VEL
LIN {X 0,Y 298.815,Z 584.718,A -85,B 0,C 180,E1 -16874.965,E2 -16874.965} C_VEL
LIN {X 0,Y 299.088,Z 587.853,A -85,B 0,C 180,E1 -16875.079,E2 -16875.079} C_VEL
LIN {X 0,Y 297.806,Z 592.286,A -85,B 0,C 180,E1 -16875.148,E2 -16875.148} C_VEL
LIN {X 0,Y 293.544,Z 601.043,A -85,B 0,C 180,E1 -16875.192,E2 -16875.192} C_VEL
LIN {X 0,Y 292.761,Z 605.075,A -85,B 0,C 180,E1 -16875.28,E2 -16875.28} C_VEL
LIN {X 0,Y 291.903,Z 645.11,A -85,B 0,C 180,E1 -16876.538,E2 -16876.538} C_VEL
LIN {X 0,Y 291.652,Z 658.54,A -85,B 0,C 180,E1 -16877.186,E2 -16877.186} C_VEL
LIN {X 0,Y 291.054,Z 671.632,A -85,B 0,C 180,E1 -16878.092,E2 -16878.092} C_VEL
LIN {X 0,Y 290.348,Z 683.6,A -85,B 0,C 180,E1 -16879.19,E2 -16879.19} C_VEL
LIN {X 0,Y 289.439,Z 695.765,A -85,B 0,C 180,E1 -16880.628,E2 -16880.628} C_VEL
LIN {X 0,Y 288.456,Z 706.812,A -85,B 0,C 180,E1 -16882.255,E2 -16882.255} C_VEL
LIN {X 0,Y 287.531,Z 716.743,A -85,B 0,C 180,E1 -16884.082,E2 -16884.082} C_VEL
LIN {X 0,Y 286.604,Z 725.982,A -85,B 0,C 180,E1 -16886.17,E2 -16886.17} C_VEL
LIN {X 0,Y 285.762,Z 734.098,A -85,B 0,C 180,E1 -16888.492,E2 -16888.492} C_VEL
LIN {X 0,Y 285.281,Z 739.667,A -85,B 0,C 180,E1 -16890.481,E2 -16890.481} C_VEL
LIN {X 0,Y 284.951,Z 744.397,A -85,B 0,C 180,E1 -16892.606,E2 -16892.606} C_VEL
LIN {X 0,Y 284.7,Z 748.659,A -85,B 0,C 180,E1 -16895.187,E2 -16895.187} C_VEL
LIN {X 0,Y 284.727,Z 750.463,A -85,B 0,C 180,E1 -16896.738,E2 -16896.738} C_VEL
LIN {X 0,Y 284.86,Z 751.795,A -85,B 0,C 180,E1 -16898.279,E2 -16898.279} C_VEL
LIN {X 0,Y 285.124,Z 752.572,A -85,B 0,C 180,E1 -16899.813,E2 -16899.813} C_VEL
LIN {X 0,Y 285.45,Z 752.894,A -85,B 0,C 180,E1 -16901.333,E2 -16901.333} C_VEL
LIN {X 0,Y 286.085,Z 752.55,A -85,B 0,C 180,E1 -16903.344,E2 -16903.344} C_VEL
LIN {X 0,Y 287.14,Z 750.953,A -85,B 0,C 180,E1 -16905.832,E2 -16905.832} C_VEL
LIN {X 0,Y 287.986,Z 749.135,A -85,B 0,C 180,E1 -16907.454,E2 -16907.454} C_VEL
LIN {X 0,Y 289.209,Z 745.995,A -85,B 0,C 180,E1 -16909.499,E2 -16909.499} C_VEL
LIN {X 0,Y 291.051,Z 740.897,A -85,B 0,C 180,E1 -16911.886,E2 -16911.886} C_VEL
LIN {X 0,Y 293.015,Z 734.45,A -85,B 0,C 180,E1 -16914.149,E2 -16914.149} C_VEL
LIN {X 0,Y 295.23,Z 726.431,A -85,B 0,C 180,E1 -16916.305,E2 -16916.305} C_VEL
LIN {X 0,Y 297.125,Z 718.732,A -85,B 0,C 180,E1 -16917.967,E2 -16917.967} C_VEL
LIN {X 0,Y 299.095,Z 709.121,A -85,B 0,C 180,E1 -16919.663,E2 -16919.663} C_VEL
LIN {X 0,Y 301.097,Z 698.283,A -85,B 0,C 180,E1 -16921.17,E2 -16921.17} C_VEL
LIN {X 0,Y 302.709,Z 686.822,A -85,B 0,C 180,E1 -16922.441,E2 -16922.441} C_VEL
LIN {X 0,Y 304.04,Z 674.573,A -85,B 0,C 180,E1 -16923.479,E2 -16923.479} C_VEL
LIN {X 0,Y 304.926,Z 661.327,A -85,B 0,C 180,E1 -16924.326,E2 -16924.326} C_VEL
LIN {X 0,Y 305.54,Z 644.083,A -85,B 0,C 180,E1 -16925.057,E2 -16925.057} C_VEL
LIN {X 0,Y 307.806,Z 606.075,A -85,B 0,C 180,E1 -16926.353,E2 -16926.353} C_VEL
LIN {X 0,Y 307.912,Z 603.106,A -85,B 0,C 180,E1 -16926.467,E2 -16926.467} C_VEL
LIN {X 0,Y 302.49,Z 593.042,A -85,B 0,C 180,E1 -16927.92,E2 -16927.92} C_VEL
LIN {X 0,Y 298.371,Z 585.821,A -85,B 0,C 180,E1 -16929.099,E2 -16929.099} C_VEL
LIN {X 0,Y 293.888,Z 579.016,A -85,B 0,C 180,E1 -16930.463,E2 -16930.463} C_VEL
LIN {X 0,Y 291.397,Z 575.303,A -85,B 0,C 180,E1 -16931.257,E2 -16931.257} C_VEL
LIN {X 0,Y 288.724,Z 571.98,A -85,B 0,C 180,E1 -16932.145,E2 -16932.145} C_VEL
LIN {X 0,Y 287.899,Z 570.275,A -85,B 0,C 180,E1 -16932.468,E2 -16932.468} C_VEL
LIN {X 0,Y 285.569,Z 568.084,A -85,B 0,C 180,E1 -16933.249,E2 -16933.249} C_VEL
LIN {X 0,Y 284.563,Z 565.681,A -85,B 0,C 180,E1 -16933.706,E2 -16933.706} C_VEL
LIN {X 0,Y 284.462,Z 565.049,A -85,B 0,C 180,E1 -16933.848,E2 -16933.848} C_VEL
LIN {X 0,Y 284.416,Z 565.059,A -85,B 0,C 180,E1 -16937.249,E2 -16937.249} C_VEL
LIN {X 0,Y 284.37,Z 565.063,A -85,B 0,C 180,E1 -16940.243,E2 -16940.243} C_VEL
LIN {X 0,Y 284.361,Z 565.064,A -85,B 0,C 180,E1 -16943.876,E2 -16943.876} C_VEL
LIN {X 0,Y 284.389,Z 565.059,A -85,B 0,C 180,E1 -16947.175,E2 -16947.175} C_VEL
LIN {X 0,Y 284.288,Z 565.073,A -85,B 0,C 180,E1 -16951.275,E2 -16951.275} C_VEL
LIN {X 0,Y 284.355,Z 565.059,A -85,B 0,C 180,E1 -16955.355,E2 -16955.355} C_VEL
LIN {X 0,Y 284.33,Z 565.091,A -85,B 0,C 180,E1 -16958.166,E2 -16958.166} C_VEL
LIN {X 0,Y 285.841,Z 569.617,A -85,B 0,C 180,E1 -16961.594,E2 -16961.594} C_VEL
LIN {X 0,Y 287.817,Z 575.029,A -85,B 0,C 180,E1 -16964.92,E2 -16964.92} C_VEL
LIN {X 0,Y 290.161,Z 582.644,A -85,B 0,C 180,E1 -16968.664,E2 -16968.664} C_VEL
LIN {X 0,Y 292.035,Z 589.72,A -85,B 0,C 180,E1 -16971.6,E2 -16971.6} C_VEL
LIN {X 0,Y 293.8,Z 597.458,A -85,B 0,C 180,E1 -16974.421,E2 -16974.421} C_VEL
LIN {X 0,Y 295.14,Z 604.496,A -85,B 0,C 180,E1 -16976.666,E2 -16976.666} C_VEL
LIN {X 0,Y 296.66,Z 609.675,A -85,B 0,C 180,E1 -16977.246,E2 -16977.246} C_VEL
LIN {X 0,Y 299.855,Z 628.444,A -85,B 0,C 180,E1 -16978.771,E2 -16978.771} C_VEL
LIN {X 0,Y 302.148,Z 646.914,A -85,B 0,C 180,E1 -16980.01,E2 -16980.01} C_VEL
LIN {X 0,Y 303.418,Z 663.029,A -85,B 0,C 180,E1 -16980.931,E2 -16980.931} C_VEL
LIN {X 0,Y 304.142,Z 682.031,A -85,B 0,C 180,E1 -16981.833,E2 -16981.833} C_VEL
LIN {X 0,Y 301.753,Z 721.555,A -85,B 0,C 180,E1 -16983.148,E2 -16983.148} C_VEL
LIN {X 0,Y 300.087,Z 735.96,A -85,B 0,C 180,E1 -16983.86,E2 -16983.86} C_VEL
LIN {X 0,Y 297.815,Z 750.159,A -85,B 0,C 180,E1 -16984.865,E2 -16984.865} C_VEL
LIN {X 0,Y 295.317,Z 762.807,A -85,B 0,C 180,E1 -16986.044,E2 -16986.044} C_VEL
LIN {X 0,Y 293.735,Z 778.178,A -85,B 0,C 180,E1 -16987.029,E2 -16987.029} C_VEL
LIN {X 0,Y 292.291,Z 790.395,A -85,B 0,C 180,E1 -16988.12,E2 -16988.12} C_VEL
LIN {X 0,Y 290.605,Z 801.879,A -85,B 0,C 180,E1 -16989.473,E2 -16989.473} C_VEL
LIN {X 0,Y 288.863,Z 812.208,A -85,B 0,C 180,E1 -16991.011,E2 -16991.011} C_VEL
LIN {X 0,Y 287.562,Z 820.672,A -85,B 0,C 180,E1 -16992.583,E2 -16992.583} C_VEL
LIN {X 0,Y 286.101,Z 828.439,A -85,B 0,C 180,E1 -16994.325,E2 -16994.325} C_VEL
LIN {X 0,Y 284.716,Z 836.009,A -85,B 0,C 180,E1 -16996.439,E2 -16996.439} C_VEL
LIN {X 0,Y 283.719,Z 842.086,A -85,B 0,C 180,E1 -16998.572,E2 -16998.572} C_VEL
LIN {X 0,Y 283.044,Z 846.889,A -85,B 0,C 180,E1 -17000.713,E2 -17000.713} C_VEL
LIN {X 0,Y 282.612,Z 850.559,A -85,B 0,C 180,E1 -17002.859,E2 -17002.859} C_VEL
LIN {X 0,Y 282.48,Z 852.555,A -85,B 0,C 180,E1 -17004.377,E2 -17004.377} C_VEL
LIN {X 0,Y 282.442,Z 854.887,A -85,B 0,C 180,E1 -17007.149,E2 -17007.149} C_VEL
LIN {X 0,Y 282.427,Z 855.502,A -85,B 0,C 180,E1 -17008.575,E2 -17008.575} C_VEL
LIN {X 0,Y 282.463,Z 855.72,A -85,B 0,C 180,E1 -17010.001,E2 -17010.001} C_VEL
LIN {X 0,Y 282.415,Z 855.493,A -85,B 0,C 180,E1 -17011.427,E2 -17011.427} C_VEL
LIN {X 0,Y 282.436,Z 854.872,A -85,B 0,C 180,E1 -17012.854,E2 -17012.854} C_VEL
LIN {X 0,Y 282.485,Z 852.516,A -85,B 0,C 180,E1 -17015.632,E2 -17015.632} C_VEL
LIN {X 0,Y 282.749,Z 849.434,A -85,B 0,C 180,E1 -17017.858,E2 -17017.858} C_VEL
LIN {X 0,Y 283.221,Z 845.385,A -85,B 0,C 180,E1 -17020.004,E2 -17020.004} C_VEL
LIN {X 0,Y 284.099,Z 839.139,A -85,B 0,C 180,E1 -17022.502,E2 -17022.502} C_VEL
LIN {X 0,Y 285.37,Z 832.333,A -85,B 0,C 180,E1 -17024.623,E2 -17024.623} C_VEL
LIN {X 0,Y 286.606,Z 825.378,A -85,B 0,C 180,E1 -17026.38,E2 -17026.38} C_VEL
LIN {X 0,Y 287.957,Z 817.286,A -85,B 0,C 180,E1 -17028.069,E2 -17028.069} C_VEL
LIN {X 0,Y 289.553,Z 807.732,A -85,B 0,C 180,E1 -17029.681,E2 -17029.681} C_VEL
LIN {X 0,Y 291.401,Z 796.261,A -85,B 0,C 180,E1 -17031.21,E2 -17031.21} C_VEL
LIN {X 0,Y 292.931,Z 784.93,A -85,B 0,C 180,E1 -17032.389,E2 -17032.389} C_VEL
LIN {X 0,Y 294.358,Z 771.935,A -85,B 0,C 180,E1 -17033.387,E2 -17033.387} C_VEL
LIN {X 0,Y 295.508,Z 758.845,A -85,B 0,C 180,E1 -17034.082,E2 -17034.082} C_VEL
LIN {X 0,Y 296.23,Z 744.203,A -85,B 0,C 180,E1 -17034.532,E2 -17034.532} C_VEL
LIN {X 0,Y 297.674,Z 682.089,A -85,B 0,C 180,E1 -17036.02,E2 -17036.02} C_VEL
LIN {X 0,Y 294.602,Z 652.671,A -85,B 0,C 180,E1 -17037.093,E2 -17037.093} C_VEL
LIN {X 0,Y 292.209,Z 635.034,A -85,B 0,C 180,E1 -17037.825,E2 -17037.825} C_VEL
LIN {X 0,Y 291.057,Z 613.893,A -85,B 0,C 180,E1 -17039.763,E2 -17039.763} C_VEL
LIN {X 0,Y 289.998,Z 598.963,A -85,B 0,C 180,E1 -17041.099,E2 -17041.099} C_VEL
LIN {X 0,Y 290.587,Z 594.708,A -85,B 0,C 180,E1 -17042.168,E2 -17042.168} C_VEL
LIN {X 0,Y 288.963,Z 586.153,A -85,B 0,C 180,E1 -17044.509,E2 -17044.509} C_VEL
LIN {X 0,Y 285.802,Z 571.631,A -85,B 0,C 180,E1 -17048.671,E2 -17048.671} C_VEL
LIN {X 0,Y 284.345,Z 565.067,A -85,B 0,C 180,E1 -17050.66,E2 -17050.66} C_VEL
LIN {X 0,Y 284.268,Z 565.063,A -85,B 0,C 180,E1 -17054.195,E2 -17054.195} C_VEL
LIN {X 0,Y 284.274,Z 565.06,A -85,B 0,C 180,E1 -17058.125,E2 -17058.125} C_VEL
LIN {X 0,Y 284.321,Z 565.059,A -85,B 0,C 180,E1 -17062.279,E2 -17062.279} C_VEL
LIN {X 0,Y 284.311,Z 565.067,A -85,B 0,C 180,E1 -17065.351,E2 -17065.351} C_VEL
LIN {X 0,Y 284.297,Z 565.052,A -85,B 0,C 180,E1 -17068.726,E2 -17068.726} C_VEL
LIN {X 0,Y 284.399,Z 565.058,A -85,B 0,C 180,E1 -17072.827,E2 -17072.827} C_VEL
LIN {X 0,Y 284.335,Z 565.055,A -85,B 0,C 180,E1 -17076.704,E2 -17076.704} C_VEL
LIN {X 0,Y 284.404,Z 565.036,A -85,B 0,C 180,E1 -17081.262,E2 -17081.262} C_VEL
LIN {X 0,Y 284.48,Z 565.044,A -85,B 0,C 180,E1 -17084.47,E2 -17084.47} C_VEL
LIN {X 0,Y 284.489,Z 565.025,A -85,B 0,C 180,E1 -17088.602,E2 -17088.602} C_VEL
LIN {X 0,Y 284.641,Z 565.015,A -85,B 0,C 180,E1 -17091.481,E2 -17091.481} C_VEL
LIN {X 0,Y 284.599,Z 565.031,A -85,B 0,C 180,E1 -17094.331,E2 -17094.331} C_VEL
LIN {X 0,Y 284.856,Z 564.982,A -85,B 0,C 180,E1 -17098.586,E2 -17098.586} C_VEL
LIN {X 0,Y 284.857,Z 565.003,A -85,B 0,C 180,E1 -17101.414,E2 -17101.414} C_VEL
LIN {X 0,Y 284.696,Z 565.013,A -85,B 0,C 180,E1 -17107.09,E2 -17107.09} C_VEL
LIN {X 0,Y 284.569,Z 565.032,A -85,B 0,C 180,E1 -17109.955,E2 -17109.955} C_VEL
LIN {X 0,Y 284.48,Z 565.038,A -85,B 0,C 180,E1 -17114.303,E2 -17114.303} C_VEL
LIN {X 0,Y 284.427,Z 565.05,A -85,B 0,C 180,E1 -17117.248,E2 -17117.248} C_VEL
LIN {X 0,Y 284.381,Z 565.043,A -85,B 0,C 180,E1 -17120.242,E2 -17120.242} C_VEL
LIN {X 0,Y 284.371,Z 565.053,A -85,B 0,C 180,E1 -17123.875,E2 -17123.875} C_VEL
LIN {X 0,Y 284.397,Z 565.056,A -85,B 0,C 180,E1 -17127.172,E2 -17127.172} C_VEL
LIN {X 0,Y 284.296,Z 565.058,A -85,B 0,C 180,E1 -17131.274,E2 -17131.274} C_VEL
LIN {X 0,Y 284.344,Z 565.056,A -85,B 0,C 180,E1 -17135.348,E2 -17135.348} C_VEL
LIN {X 0,Y 284.325,Z 565.071,A -85,B 0,C 180,E1 -17138.167,E2 -17138.167} C_VEL
LIN {X 0,Y 284.272,Z 565.074,A -85,B 0,C 180,E1 -17142.124,E2 -17142.124} C_VEL
LIN {X 0,Y 284.258,Z 565.058,A -85,B 0,C 180,E1 -17146.189,E2 -17146.189} C_VEL
LIN {X 0,Y 284.32,Z 565.198,A -85,B 0,C 180,E1 -17148.689,E2 -17148.689} C_VEL
LIN {X 0,Y 288.745,Z 578.567,A -85,B 0,C 180,E1 -17152.28,E2 -17152.28} C_VEL
LIN {X 0,Y 292.066,Z 590.577,A -85,B 0,C 180,E1 -17155.255,E2 -17155.255} C_VEL
LIN {X 0,Y 294.817,Z 602.502,A -85,B 0,C 180,E1 -17158.043,E2 -17158.043} C_VEL
LIN {X 0,Y 295.549,Z 606.288,A -85,B 0,C 180,E1 -17158.878,E2 -17158.878} C_VEL
LIN {X 0,Y 294.084,Z 622.122,A -85,B 0,C 180,E1 -17161.736,E2 -17161.736} C_VEL
LIN {X 0,Y 293.842,Z 625.163,A -85,B 0,C 180,E1 -17162.266,E2 -17162.266} C_VEL
LIN {X 0,Y 298.304,Z 652.831,A -85,B 0,C 180,E1 -17163.461,E2 -17163.461} C_VEL
LIN {X 0,Y 298.891,Z 658.073,A -85,B 0,C 180,E1 -17163.656,E2 -17163.656} C_VEL
LIN {X 0,Y 296.715,Z 736.685,A -85,B 0,C 180,E1 -17165.558,E2 -17165.558} C_VEL
LIN {X 0,Y 295.959,Z 749.499,A -85,B 0,C 180,E1 -17166.097,E2 -17166.097} C_VEL
LIN {X 0,Y 294.967,Z 761.276,A -85,B 0,C 180,E1 -17166.849,E2 -17166.849} C_VEL
LIN {X 0,Y 293.797,Z 771.213,A -85,B 0,C 180,E1 -17167.681,E2 -17167.681} C_VEL
LIN {X 0,Y 292.056,Z 783.522,A -85,B 0,C 180,E1 -17169.025,E2 -17169.025} C_VEL
LIN {X 0,Y 290.469,Z 794.199,A -85,B 0,C 180,E1 -17170.529,E2 -17170.529} C_VEL
LIN {X 0,Y 288.868,Z 804.085,A -85,B 0,C 180,E1 -17172.294,E2 -17172.294} C_VEL
LIN {X 0,Y 287.046,Z 813.464,A -85,B 0,C 180,E1 -17174.375,E2 -17174.375} C_VEL
LIN {X 0,Y 285.62,Z 820.915,A -85,B 0,C 180,E1 -17176.481,E2 -17176.481} C_VEL
LIN {X 0,Y 284.456,Z 826.898,A -85,B 0,C 180,E1 -17178.599,E2 -17178.599} C_VEL
LIN {X 0,Y 283.602,Z 831.626,A -85,B 0,C 180,E1 -17180.73,E2 -17180.73} C_VEL
LIN {X 0,Y 283.053,Z 835.237,A -85,B 0,C 180,E1 -17182.867,E2 -17182.867} C_VEL
LIN {X 0,Y 282.765,Z 837.098,A -85,B 0,C 180,E1 -17184.293,E2 -17184.293} C_VEL
LIN {X 0,Y 282.613,Z 838.516,A -85,B 0,C 180,E1 -17185.72,E2 -17185.72} C_VEL
LIN {X 0,Y 282.482,Z 839.511,A -85,B 0,C 180,E1 -17187.147,E2 -17187.147} C_VEL
LIN {X 0,Y 282.362,Z 840.358,A -85,B 0,C 180,E1 -17189.999,E2 -17189.999} C_VEL
LIN {X 0,Y 282.375,Z 840.164,A -85,B 0,C 180,E1 -17191.425,E2 -17191.425} C_VEL
LIN {X 0,Y 282.478,Z 839.575,A -85,B 0,C 180,E1 -17192.851,E2 -17192.851} C_VEL
LIN {X 0,Y 282.608,Z 838.606,A -85,B 0,C 180,E1 -17194.277,E2 -17194.277} C_VEL
LIN {X 0,Y 282.894,Z 836.369,A -85,B 0,C 180,E1 -17196.417,E2 -17196.417} C_VEL
LIN {X 0,Y 283.364,Z 833.155,A -85,B 0,C 180,E1 -17198.557,E2 -17198.557} C_VEL
LIN {X 0,Y 284.092,Z 828.877,A -85,B 0,C 180,E1 -17200.691,E2 -17200.691} C_VEL
LIN {X 0,Y 285.133,Z 823.413,A -85,B 0,C 180,E1 -17202.815,E2 -17202.815} C_VEL
LIN {X 0,Y 286.448,Z 816.554,A -85,B 0,C 180,E1 -17204.927,E2 -17204.927} C_VEL
LIN {X 0,Y 288.179,Z 807.956,A -85,B 0,C 180,E1 -17207.015,E2 -17207.015} C_VEL
LIN {X 0,Y 289.756,Z 798.952,A -85,B 0,C 180,E1 -17208.783,E2 -17208.783} C_VEL
LIN {X 0,Y 291.426,Z 788.218,A -85,B 0,C 180,E1 -17210.466,E2 -17210.466} C_VEL
LIN {X 0,Y 293.078,Z 777.205,A -85,B 0,C 180,E1 -17211.818,E2 -17211.818} C_VEL
LIN {X 0,Y 294.391,Z 766.788,A -85,B 0,C 180,E1 -17212.824,E2 -17212.824} C_VEL
LIN {X 0,Y 295.577,Z 754.228,A -85,B 0,C 180,E1 -17213.747,E2 -17213.747} C_VEL
LIN {X 0,Y 296.518,Z 740.869,A -85,B 0,C 180,E1 -17214.411,E2 -17214.411} C_VEL
LIN {X 0,Y 297.095,Z 724.73,A -85,B 0,C 180,E1 -17214.873,E2 -17214.873} C_VEL
LIN {X 0,Y 298.804,Z 659.461,A -85,B 0,C 180,E1 -17216.433,E2 -17216.433} C_VEL
LIN {X 0,Y 294.648,Z 634.829,A -85,B 0,C 180,E1 -17217.5,E2 -17217.5} C_VEL
LIN {X 0,Y 292.983,Z 625.787,A -85,B 0,C 180,E1 -17217.965,E2 -17217.965} C_VEL
LIN {X 0,Y 294.762,Z 607.524,A -85,B 0,C 180,E1 -17221.636,E2 -17221.636} C_VEL
LIN {X 0,Y 294.606,Z 604.2,A -85,B 0,C 180,E1 -17222.391,E2 -17222.391} C_VEL
LIN {X 0,Y 292.297,Z 592.952,A -85,B 0,C 180,E1 -17225.242,E2 -17225.242} C_VEL
LIN {X 0,Y 289.752,Z 582.788,A -85,B 0,C 180,E1 -17227.993,E2 -17227.993} C_VEL
LIN {X 0,Y 286.477,Z 571.822,A -85,B 0,C 180,E1 -17231.099,E2 -17231.099} C_VEL
LIN {X 0,Y 284.335,Z 565.045,A -85,B 0,C 180,E1 -17233.178,E2 -17233.178} C_VEL
LIN {X 0,Y 284.368,Z 565.27,A -85,B 0,C 180,E1 -17233.45,E2 -17233.45} C_VEL
LIN {X 0,Y 293.316,Z 590.086,A -85,B 0,C 180,E1 -17234.826,E2 -17234.826} C_VEL
LIN {X 0,Y 292.761,Z 605.075,A -85,B 0,C 180,E1 -17235.28,E2 -17235.28} C_VEL
LIN {X 0,Y 292.029,Z 610.885,A -85,B 0,C 180,E1 -17235.43,E2 -17235.43} C_VEL
LIN {X 0,Y 285.847,Z 629.713,A -85,B 0,C 180,E1 -17235.708,E2 -17235.708} C_VEL
LIN {X 0,Y 285.125,Z 635.526,A -85,B 0,C 180,E1 -17235.862,E2 -17235.862} C_VEL
LIN {X 0,Y 284.94,Z 652.813,A -85,B 0,C 180,E1 -17236.519,E2 -17236.519} C_VEL
LIN {X 0,Y 284.49,Z 665.617,A -85,B 0,C 180,E1 -17237.284,E2 -17237.284} C_VEL
LIN {X 0,Y 283.78,Z 679.133,A -85,B 0,C 180,E1 -17238.392,E2 -17238.392} C_VEL
LIN {X 0,Y 282.89,Z 691.728,A -85,B 0,C 180,E1 -17239.764,E2 -17239.764} C_VEL
LIN {X 0,Y 281.957,Z 702.762,A -85,B 0,C 180,E1 -17241.271,E2 -17241.271} C_VEL
LIN {X 0,Y 281.049,Z 712.412,A -85,B 0,C 180,E1 -17242.895,E2 -17242.895} C_VEL
LIN {X 0,Y 280.114,Z 721.481,A -85,B 0,C 180,E1 -17244.755,E2 -17244.755} C_VEL
LIN {X 0,Y 279.278,Z 729.678,A -85,B 0,C 180,E1 -17246.815,E2 -17246.815} C_VEL
LIN {X 0,Y 278.538,Z 736.922,A -85,B 0,C 180,E1 -17249.075,E2 -17249.075} C_VEL
LIN {X 0,Y 278.108,Z 742.56,A -85,B 0,C 180,E1 -17251.305,E2 -17251.305} C_VEL
LIN {X 0,Y 277.775,Z 747.277,A -85,B 0,C 180,E1 -17253.719,E2 -17253.719} C_VEL
LIN {X 0,Y 277.673,Z 750.677,A -85,B 0,C 180,E1 -17256.111,E2 -17256.111} C_VEL
LIN {X 0,Y 277.757,Z 752.254,A -85,B 0,C 180,E1 -17257.695,E2 -17257.695} C_VEL
LIN {X 0,Y 277.984,Z 753.332,A -85,B 0,C 180,E1 -17259.293,E2 -17259.293} C_VEL
LIN {X 0,Y 278.328,Z 753.915,A -85,B 0,C 180,E1 -17260.837,E2 -17260.837} C_VEL
LIN {X 0,Y 279.011,Z 753.857,A -85,B 0,C 180,E1 -17263.165,E2 -17263.165} C_VEL
LIN {X 0,Y 279.953,Z 752.735,A -85,B 0,C 180,E1 -17265.461,E2 -17265.461} C_VEL
LIN {X 0,Y 280.936,Z 751.021,A -85,B 0,C 180,E1 -17267.318,E2 -17267.318} C_VEL
LIN {X 0,Y 282.086,Z 748.446,A -85,B 0,C 180,E1 -17269.23,E2 -17269.23} C_VEL
LIN {X 0,Y 283.768,Z 744.325,A -85,B 0,C 180,E1 -17271.454,E2 -17271.454} C_VEL
LIN {X 0,Y 285.637,Z 738.944,A -85,B 0,C 180,E1 -17273.643,E2 -17273.643} C_VEL
LIN {X 0,Y 287.753,Z 732.097,A -85,B 0,C 180,E1 -17275.798,E2 -17275.798} C_VEL
LIN {X 0,Y 290.171,Z 723.506,A -85,B 0,C 180,E1 -17277.918,E2 -17277.918} C_VEL
LIN {X 0,Y 292.448,Z 713.669,A -85,B 0,C 180,E1 -17279.828,E2 -17279.828} C_VEL
LIN {X 0,Y 294.508,Z 703.662,A -85,B 0,C 180,E1 -17281.367,E2 -17281.367} C_VEL
LIN {X 0,Y 296.347,Z 692.75,A -85,B 0,C 180,E1 -17282.719,E2 -17282.719} C_VEL
LIN {X 0,Y 297.849,Z 681.52,A -85,B 0,C 180,E1 -17283.816,E2 -17283.816} C_VEL
LIN {X 0,Y 299.092,Z 668.347,A -85,B 0,C 180,E1 -17284.802,E2 -17284.802} C_VEL
LIN {X 0,Y 299.776,Z 654.377,A -85,B 0,C 180,E1 -17285.536,E2 -17285.536} C_VEL
LIN {X 0,Y 301.217,Z 625.269,A -85,B 0,C 180,E1 -17286.611,E2 -17286.611} C_VEL
LIN {X 0,Y 302.576,Z 605.856,A -85,B 0,C 180,E1 -17287.286,E2 -17287.286} C_VEL
LIN {X 0,Y 294.951,Z 591.707,A -85,B 0,C 180,E1 -17289.529,E2 -17289.529} C_VEL
LIN {X 0,Y 290.155,Z 584.372,A -85,B 0,C 180,E1 -17291.035,E2 -17291.035} C_VEL
LIN {X 0,Y 287.265,Z 580.165,A -85,B 0,C 180,E1 -17292.03,E2 -17292.03} C_VEL
LIN {X 0,Y 284.924,Z 576.748,A -85,B 0,C 180,E1 -17292.872,E2 -17292.872} C_VEL
LIN {X 0,Y 281.96,Z 573.038,A -85,B 0,C 180,E1 -17293.99,E2 -17293.99} C_VEL
LIN {X 0,Y 281.077,Z 571.287,A -85,B 0,C 180,E1 -17294.387,E2 -17294.387} C_VEL
LIN {X 0,Y 278.673,Z 569.13,A -85,B 0,C 180,E1 -17295.327,E2 -17295.327} C_VEL
LIN {X 0,Y 277.56,Z 566.609,A -85,B 0,C 180,E1 -17295.909,E2 -17295.909} C_VEL
LIN {X 0,Y 277.418,Z 565.92,A -85,B 0,C 180,E1 -17296.053,E2 -17296.053} C_VEL
LIN {X 0,Y 277.336,Z 565.94,A -85,B 0,C 180,E1 -17300.35,E2 -17300.35} C_VEL
LIN {X 0,Y 277.311,Z 565.941,A -85,B 0,C 180,E1 -17304.171,E2 -17304.171} C_VEL
LIN {X 0,Y 277.318,Z 565.939,A -85,B 0,C 180,E1 -17307.506,E2 -17307.506} C_VEL
LIN {X 0,Y 277.264,Z 565.947,A -85,B 0,C 180,E1 -17310.482,E2 -17310.482} C_VEL
LIN {X 0,Y 277.292,Z 565.953,A -85,B 0,C 180,E1 -17314.99,E2 -17314.99} C_VEL
LIN {X 0,Y 278.722,Z 570.195,A -85,B 0,C 180,E1 -17319.078,E2 -17319.078} C_VEL
LIN {X 0,Y 280.491,Z 574.938,A -85,B 0,C 180,E1 -17322.572,E2 -17322.572} C_VEL
LIN {X 0,Y 282.322,Z 580.503,A -85,B 0,C 180,E1 -17325.814,E2 -17325.814} C_VEL
LIN {X 0,Y 284.192,Z 586.961,A -85,B 0,C 180,E1 -17328.961,E2 -17328.961} C_VEL
LIN {X 0,Y 286.105,Z 594.53,A -85,B 0,C 180,E1 -17332.115,E2 -17332.115} C_VEL
LIN {X 0,Y 287.818,Z 602.298,A -85,B 0,C 180,E1 -17334.885,E2 -17334.885} C_VEL
LIN {X 0,Y 290.629,Z 608.525,A -85,B 0,C 180,E1 -17335.898,E2 -17335.898} C_VEL
LIN {X 0,Y 291.884,Z 612.644,A -85,B 0,C 180,E1 -17336.398,E2 -17336.398} C_VEL
LIN {X 0,Y 294.885,Z 631.506,A -85,B 0,C 180,E1 -17337.973,E2 -17337.973} C_VEL
LIN {X 0,Y 296.846,Z 648.363,A -85,B 0,C 180,E1 -17339.151,E2 -17339.151} C_VEL
LIN {X 0,Y 298.074,Z 665.274,A -85,B 0,C 180,E1 -17340.143,E2 -17340.143} C_VEL
LIN {X 0,Y 298.535,Z 684.394,A -85,B 0,C 180,E1 -17341.077,E2 -17341.077} C_VEL
LIN {X 0,Y 296.161,Z 720.383,A -85,B 0,C 180,E1 -17342.294,E2 -17342.294} C_VEL
LIN {X 0,Y 294.392,Z 734.966,A -85,B 0,C 180,E1 -17343.028,E2 -17343.028} C_VEL
LIN {X 0,Y 292.172,Z 748.088,A -85,B 0,C 180,E1 -17343.962,E2 -17343.962} C_VEL
LIN {X 0,Y 289.724,Z 760.044,A -85,B 0,C 180,E1 -17345.074,E2 -17345.074} C_VEL
LIN {X 0,Y 288.515,Z 765.968,A -85,B 0,C 180,E1 -17345.682,E2 -17345.682} C_VEL
LIN {X 0,Y 287.088,Z 779.127,A -85,B 0,C 180,E1 -17346.561,E2 -17346.561} C_VEL
LIN {X 0,Y 285.701,Z 790.223,A -85,B 0,C 180,E1 -17347.588,E2 -17347.588} C_VEL
LIN {X 0,Y 283.958,Z 801.701,A -85,B 0,C 180,E1 -17348.97,E2 -17348.97} C_VEL
LIN {X 0,Y 282.142,Z 812.026,A -85,B 0,C 180,E1 -17350.541,E2 -17350.541} C_VEL
LIN {X 0,Y 280.658,Z 821.14,A -85,B 0,C 180,E1 -17352.285,E2 -17352.285} C_VEL
LIN {X 0,Y 279.005,Z 829.607,A -85,B 0,C 180,E1 -17354.29,E2 -17354.29} C_VEL
LIN {X 0,Y 277.563,Z 836.933,A -85,B 0,C 180,E1 -17356.456,E2 -17356.456} C_VEL
LIN {X 0,Y 276.71,Z 841.894,A -85,B 0,C 180,E1 -17358.278,E2 -17358.278} C_VEL
LIN {X 0,Y 276.001,Z 846.697,A -85,B 0,C 180,E1 -17360.474,E2 -17360.474} C_VEL
LIN {X 0,Y 275.539,Z 850.367,A -85,B 0,C 180,E1 -17362.674,E2 -17362.674} C_VEL
LIN {X 0,Y 275.375,Z 852.604,A -85,B 0,C 180,E1 -17364.468,E2 -17364.468} C_VEL
LIN {X 0,Y 275.348,Z 854.694,A -85,B 0,C 180,E1 -17367.075,E2 -17367.075} C_VEL
LIN {X 0,Y 275.348,Z 855.309,A -85,B 0,C 180,E1 -17368.539,E2 -17368.539} C_VEL
LIN {X 0,Y 275.38,Z 855.527,A -85,B 0,C 180,E1 -17370.001,E2 -17370.001} C_VEL
LIN {X 0,Y 275.337,Z 855.3,A -85,B 0,C 180,E1 -17371.464,E2 -17371.464} C_VEL
LIN {X 0,Y 275.343,Z 854.679,A -85,B 0,C 180,E1 -17372.927,E2 -17372.927} C_VEL
LIN {X 0,Y 275.408,Z 852.51,A -85,B 0,C 180,E1 -17375.601,E2 -17375.601} C_VEL
LIN {X 0,Y 275.707,Z 849.241,A -85,B 0,C 180,E1 -17378.061,E2 -17378.061} C_VEL
LIN {X 0,Y 276.201,Z 845.191,A -85,B 0,C 180,E1 -17380.261,E2 -17380.261} C_VEL
LIN {X 0,Y 277.143,Z 838.945,A -85,B 0,C 180,E1 -17382.821,E2 -17382.821} C_VEL
LIN {X 0,Y 278.493,Z 832.141,A -85,B 0,C 180,E1 -17384.992,E2 -17384.992} C_VEL
LIN {X 0,Y 279.791,Z 825.187,A -85,B 0,C 180,E1 -17386.791,E2 -17386.791} C_VEL
LIN {X 0,Y 281.257,Z 816.79,A -85,B 0,C 180,E1 -17388.578,E2 -17388.578} C_VEL
LIN {X 0,Y 283.066,Z 806.381,A -85,B 0,C 180,E1 -17390.341,E2 -17390.341} C_VEL
LIN {X 0,Y 285.004,Z 794.655,A -85,B 0,C 180,E1 -17391.9,E2 -17391.9} C_VEL
LIN {X 0,Y 286.621,Z 782.807,A -85,B 0,C 180,E1 -17393.1,E2 -17393.1} C_VEL
LIN {X 0,Y 287.995,Z 770.493,A -85,B 0,C 180,E1 -17394.032,E2 -17394.032} C_VEL
LIN {X 0,Y 289.13,Z 757.655,A -85,B 0,C 180,E1 -17394.696,E2 -17394.696} C_VEL
LIN {X 0,Y 289.829,Z 742.306,A -85,B 0,C 180,E1 -17395.159,E2 -17395.159} C_VEL
LIN {X 0,Y 291.306,Z 683.085,A -85,B 0,C 180,E1 -17396.603,E2 -17396.603} C_VEL
LIN {X 0,Y 288.413,Z 654.511,A -85,B 0,C 180,E1 -17397.671,E2 -17397.671} C_VEL
LIN {X 0,Y 285.764,Z 634.878,A -85,B 0,C 180,E1 -17398.508,E2 -17398.508} C_VEL
LIN {X 0,Y 284.575,Z 611.155,A -85,B 0,C 180,E1 -17400.764,E2 -17400.764} C_VEL
LIN {X 0,Y 283.534,Z 596.067,A -85,B 0,C 180,E1 -17402.198,E2 -17402.198} C_VEL
LIN {X 0,Y 282.759,Z 591.072,A -85,B 0,C 180,E1 -17403.576,E2 -17403.576} C_VEL
LIN {X 0,Y 280.009,Z 578.394,A -85,B 0,C 180,E1 -17407.247,E2 -17407.247} C_VEL
LIN {X 0,Y 277.264,Z 565.949,A -85,B 0,C 180,E1 -17411.02,E2 -17411.02} C_VEL
LIN {X 0,Y 277.22,Z 565.947,A -85,B 0,C 180,E1 -17415.223,E2 -17415.223} C_VEL
LIN {X 0,Y 277.224,Z 565.944,A -85,B 0,C 180,E1 -17419.513,E2 -17419.513} C_VEL
LIN {X 0,Y 277.267,Z 565.934,A -85,B 0,C 180,E1 -17422.53,E2 -17422.53} C_VEL
LIN {X 0,Y 277.249,Z 565.949,A -85,B 0,C 180,E1 -17426.105,E2 -17426.105} C_VEL
LIN {X 0,Y 277.264,Z 565.929,A -85,B 0,C 180,E1 -17429.539,E2 -17429.539} C_VEL
LIN {X 0,Y 277.361,Z 565.934,A -85,B 0,C 180,E1 -17432.864,E2 -17432.864} C_VEL
LIN {X 0,Y 277.299,Z 565.923,A -85,B 0,C 180,E1 -17436.077,E2 -17436.077} C_VEL
LIN {X 0,Y 277.346,Z 565.92,A -85,B 0,C 180,E1 -17440.766,E2 -17440.766} C_VEL
LIN {X 0,Y 277.43,Z 565.926,A -85,B 0,C 180,E1 -17445.326,E2 -17445.326} C_VEL
LIN {X 0,Y 277.463,Z 565.894,A -85,B 0,C 180,E1 -17449.787,E2 -17449.787} C_VEL
LIN {X 0,Y 277.643,Z 565.898,A -85,B 0,C 180,E1 -17452.729,E2 -17452.729} C_VEL
LIN {X 0,Y 277.822,Z 565.856,A -85,B 0,C 180,E1 -17458.551,E2 -17458.551} C_VEL
LIN {X 0,Y 277.823,Z 565.88,A -85,B 0,C 180,E1 -17461.45,E2 -17461.45} C_VEL
LIN {X 0,Y 277.651,Z 565.891,A -85,B 0,C 180,E1 -17467.271,E2 -17467.271} C_VEL
LIN {X 0,Y 277.509,Z 565.91,A -85,B 0,C 180,E1 -17470.211,E2 -17470.211} C_VEL
LIN {X 0,Y 277.43,Z 565.922,A -85,B 0,C 180,E1 -17474.674,E2 -17474.674} C_VEL
LIN {X 0,Y 277.347,Z 565.914,A -85,B 0,C 180,E1 -17479.234,E2 -17479.234} C_VEL
LIN {X 0,Y 277.321,Z 565.928,A -85,B 0,C 180,E1 -17484.17,E2 -17484.17} C_VEL
LIN {X 0,Y 277.325,Z 565.938,A -85,B 0,C 180,E1 -17487.504,E2 -17487.504} C_VEL
LIN {X 0,Y 277.275,Z 565.931,A -85,B 0,C 180,E1 -17490.481,E2 -17490.481} C_VEL
LIN {X 0,Y 277.25,Z 565.95,A -85,B 0,C 180,E1 -17493.896,E2 -17493.896} C_VEL
LIN {X 0,Y 277.282,Z 565.949,A -85,B 0,C 180,E1 -17497.467,E2 -17497.467} C_VEL
LIN {X 0,Y 277.213,Z 565.957,A -85,B 0,C 180,E1 -17501.236,E2 -17501.236} C_VEL
LIN {X 0,Y 277.203,Z 565.953,A -85,B 0,C 180,E1 -17505.226,E2 -17505.226} C_VEL
LIN {X 0,Y 277.254,Z 566.082,A -85,B 0,C 180,E1 -17507.731,E2 -17507.731} C_VEL
LIN {X 0,Y 281.376,Z 578.151,A -85,B 0,C 180,E1 -17511.118,E2 -17511.118} C_VEL
LIN {X 0,Y 284.669,Z 589.301,A -85,B 0,C 180,E1 -17514.003,E2 -17514.003} C_VEL
LIN {X 0,Y 287.92,Z 602.925,A -85,B 0,C 180,E1 -17517.273,E2 -17517.273} C_VEL
LIN {X 0,Y 288.995,Z 608.384,A -85,B 0,C 180,E1 -17518.512,E2 -17518.512} C_VEL
LIN {X 0,Y 287.658,Z 622.422,A -85,B 0,C 180,E1 -17521.082,E2 -17521.082} C_VEL
LIN {X 0,Y 287.455,Z 625.756,A -85,B 0,C 180,E1 -17521.617,E2 -17521.617} C_VEL
LIN {X 0,Y 291.729,Z 652.173,A -85,B 0,C 180,E1 -17522.794,E2 -17522.794} C_VEL
LIN {X 0,Y 292.53,Z 658.349,A -85,B 0,C 180,E1 -17523.042,E2 -17523.042} C_VEL
LIN {X 0,Y 290.234,Z 738.132,A -85,B 0,C 180,E1 -17525.023,E2 -17525.023} C_VEL
LIN {X 0,Y 289.356,Z 751.156,A -85,B 0,C 180,E1 -17525.612,E2 -17525.612} C_VEL
LIN {X 0,Y 288.027,Z 764.673,A -85,B 0,C 180,E1 -17526.544,E2 -17526.544} C_VEL
LIN {X 0,Y 286.583,Z 776.413,A -85,B 0,C 180,E1 -17527.658,E2 -17527.658} C_VEL
LIN {X 0,Y 284.835,Z 787.606,A -85,B 0,C 180,E1 -17529.036,E2 -17529.036} C_VEL
LIN {X 0,Y 283.159,Z 798.104,A -85,B 0,C 180,E1 -17530.68,E2 -17530.68} C_VEL
LIN {X 0,Y 281.791,Z 806.01,A -85,B 0,C 180,E1 -17532.21,E2 -17532.21} C_VEL
LIN {X 0,Y 279.907,Z 814.991,A -85,B 0,C 180,E1 -17534.34,E2 -17534.34} C_VEL
LIN {X 0,Y 278.492,Z 822.199,A -85,B 0,C 180,E1 -17536.5,E2 -17536.5} C_VEL
LIN {X 0,Y 277.141,Z 828.814,A -85,B 0,C 180,E1 -17539.035,E2 -17539.035} C_VEL
LIN {X 0,Y 276.367,Z 833.151,A -85,B 0,C 180,E1 -17541.222,E2 -17541.222} C_VEL
LIN {X 0,Y 275.78,Z 836.712,A -85,B 0,C 180,E1 -17543.661,E2 -17543.661} C_VEL
LIN {X 0,Y 275.539,Z 838.709,A -85,B 0,C 180,E1 -17545.61,E2 -17545.61} C_VEL
LIN {X 0,Y 275.416,Z 839.703,A -85,B 0,C 180,E1 -17547.073,E2 -17547.073} C_VEL
LIN {X 0,Y 275.284,Z 840.55,A -85,B 0,C 180,E1 -17549.999,E2 -17549.999} C_VEL
LIN {X 0,Y 275.301,Z 840.356,A -85,B 0,C 180,E1 -17551.462,E2 -17551.462} C_VEL
LIN {X 0,Y 275.413,Z 839.767,A -85,B 0,C 180,E1 -17552.924,E2 -17552.924} C_VEL
LIN {X 0,Y 275.536,Z 838.799,A -85,B 0,C 180,E1 -17554.387,E2 -17554.387} C_VEL
LIN {X 0,Y 275.783,Z 836.844,A -85,B 0,C 180,E1 -17556.345,E2 -17556.345} C_VEL
LIN {X 0,Y 276.327,Z 833.347,A -85,B 0,C 180,E1 -17558.776,E2 -17558.776} C_VEL
LIN {X 0,Y 277.108,Z 829.068,A -85,B 0,C 180,E1 -17560.964,E2 -17560.964} C_VEL
LIN {X 0,Y 278.206,Z 823.602,A -85,B 0,C 180,E1 -17563.14,E2 -17563.14} C_VEL
LIN {X 0,Y 279.569,Z 816.742,A -85,B 0,C 180,E1 -17565.303,E2 -17565.303} C_VEL
LIN {X 0,Y 281.387,Z 808.142,A -85,B 0,C 180,E1 -17567.439,E2 -17567.439} C_VEL
LIN {X 0,Y 283.001,Z 799.235,A -85,B 0,C 180,E1 -17569.229,E2 -17569.229} C_VEL
LIN {X 0,Y 284.789,Z 788.395,A -85,B 0,C 180,E1 -17570.965,E2 -17570.965} C_VEL
LIN {X 0,Y 286.502,Z 777.377,A -85,B 0,C 180,E1 -17572.346,E2 -17572.346} C_VEL
LIN {X 0,Y 287.983,Z 765.995,A -85,B 0,C 180,E1 -17573.457,E2 -17573.457} C_VEL
LIN {X 0,Y 289.219,Z 752.952,A -85,B 0,C 180,E1 -17574.398,E2 -17574.398} C_VEL
LIN {X 0,Y 290.153,Z 739.957,A -85,B 0,C 180,E1 -17575.03,E2 -17575.03} C_VEL
LIN {X 0,Y 290.891,Z 719.446,A -85,B 0,C 180,E1 -17575.584,E2 -17575.584} C_VEL
LIN {X 0,Y 292.486,Z 660.647,A -85,B 0,C 180,E1 -17577.019,E2 -17577.019} C_VEL
LIN {X 0,Y 288.78,Z 638.219,A -85,B 0,C 180,E1 -17578.015,E2 -17578.015} C_VEL
LIN {X 0,Y 286.512,Z 625.896,A -85,B 0,C 180,E1 -17578.648,E2 -17578.648} C_VEL
LIN {X 0,Y 288.223,Z 609.236,A -85,B 0,C 180,E1 -17582.053,E2 -17582.053} C_VEL
LIN {X 0,Y 287.622,Z 604.074,A -85,B 0,C 180,E1 -17583.294,E2 -17583.294} C_VEL
LIN {X 0,Y 285.173,Z 592.728,A -85,B 0,C 180,E1 -17586.259,E2 -17586.259} C_VEL
LIN {X 0,Y 282.487,Z 582.374,A -85,B 0,C 180,E1 -17589.165,E2 -17589.165} C_VEL
LIN {X 0,Y 278.996,Z 571.02,A -85,B 0,C 180,E1 -17592.54,E2 -17592.54} C_VEL
LIN {X 0,Y 278.238,Z 569.061,A -85,B 0,C 180,E1 -17593.185,E2 -17593.185} C_VEL
LIN {X 0,Y 286.452,Z 591.348,A -85,B 0,C 180,E1 -17594.467,E2 -17594.467} C_VEL
LIN {X 0,Y 285.125,Z 635.526,A -85,B 0,C 180,E1 -17595.862,E2 -17595.862} C_VEL
LIN {X 0,Y 284.433,Z 641.347,A -85,B 0,C 180,E1 -17596.019,E2 -17596.019} C_VEL
LIN {X 0,Y 281.518,Z 650.778,A -85,B 0,C 180,E1 -17596.241,E2 -17596.241} C_VEL
LIN {X 0,Y 278.491,Z 660.073,A -85,B 0,C 180,E1 -17596.58,E2 -17596.58} C_VEL
LIN {X 0,Y 277.627,Z 665.676,A -85,B 0,C 180,E1 -17596.921,E2 -17596.921} C_VEL
LIN {X 0,Y 276.854,Z 679.742,A -85,B 0,C 180,E1 -17598.091,E2 -17598.091} C_VEL
LIN {X 0,Y 275.955,Z 692.405,A -85,B 0,C 180,E1 -17599.497,E2 -17599.497} C_VEL
LIN {X 0,Y 275.017,Z 703.217,A -85,B 0,C 180,E1 -17601.002,E2 -17601.002} C_VEL
LIN {X 0,Y 274.069,Z 712.881,A -85,B 0,C 180,E1 -17602.646,E2 -17602.646} C_VEL
LIN {X 0,Y 273.093,Z 722.301,A -85,B 0,C 180,E1 -17604.617,E2 -17604.617} C_VEL
LIN {X 0,Y 272.216,Z 730.542,A -85,B 0,C 180,E1 -17606.727,E2 -17606.727} C_VEL
LIN {X 0,Y 271.528,Z 737.221,A -85,B 0,C 180,E1 -17608.824,E2 -17608.824} C_VEL
LIN {X 0,Y 271.048,Z 743.374,A -85,B 0,C 180,E1 -17611.261,E2 -17611.261} C_VEL
LIN {X 0,Y 270.731,Z 748.289,A -85,B 0,C 180,E1 -17613.812,E2 -17613.812} C_VEL
LIN {X 0,Y 270.617,Z 750.731,A -85,B 0,C 180,E1 -17615.447,E2 -17615.447} C_VEL
LIN {X 0,Y 270.673,Z 752.576,A -85,B 0,C 180,E1 -17617.078,E2 -17617.078} C_VEL
LIN {X 0,Y 270.897,Z 754.158,A -85,B 0,C 180,E1 -17619.055,E2 -17619.055} C_VEL
LIN {X 0,Y 271.593,Z 755.114,A -85,B 0,C 180,E1 -17621.909,E2 -17621.909} C_VEL
LIN {X 0,Y 272.121,Z 755.006,A -85,B 0,C 180,E1 -17623.495,E2 -17623.495} C_VEL
LIN {X 0,Y 272.78,Z 754.374,A -85,B 0,C 180,E1 -17625.07,E2 -17625.07} C_VEL
LIN {X 0,Y 273.882,Z 752.792,A -85,B 0,C 180,E1 -17627.179,E2 -17627.179} C_VEL
LIN {X 0,Y 275.43,Z 749.667,A -85,B 0,C 180,E1 -17629.711,E2 -17629.711} C_VEL
LIN {X 0,Y 277.253,Z 745.534,A -85,B 0,C 180,E1 -17632.014,E2 -17632.014} C_VEL
LIN {X 0,Y 279.228,Z 740.293,A -85,B 0,C 180,E1 -17634.222,E2 -17634.222} C_VEL
LIN {X 0,Y 281.625,Z 733.079,A -85,B 0,C 180,E1 -17636.534,E2 -17636.534} C_VEL
LIN {X 0,Y 284.052,Z 724.914,A -85,B 0,C 180,E1 -17638.582,E2 -17638.582} C_VEL
LIN {X 0,Y 286.239,Z 716.188,A -85,B 0,C 180,E1 -17640.352,E2 -17640.352} C_VEL
LIN {X 0,Y 288.577,Z 705.902,A -85,B 0,C 180,E1 -17642.006,E2 -17642.006} C_VEL
LIN {X 0,Y 290.657,Z 694.549,A -85,B 0,C 180,E1 -17643.466,E2 -17643.466} C_VEL
LIN {X 0,Y 292.325,Z 682.644,A -85,B 0,C 180,E1 -17644.654,E2 -17644.654} C_VEL
LIN {X 0,Y 293.615,Z 669.911,A -85,B 0,C 180,E1 -17645.623,E2 -17645.623} C_VEL
LIN {X 0,Y 294.37,Z 656.967,A -85,B 0,C 180,E1 -17646.34,E2 -17646.34} C_VEL
LIN {X 0,Y 295.832,Z 629.113,A -85,B 0,C 180,E1 -17647.425,E2 -17647.425} C_VEL
LIN {X 0,Y 297.301,Z 608.672,A -85,B 0,C 180,E1 -17648.154,E2 -17648.154} C_VEL
LIN {X 0,Y 290.841,Z 596.427,A -85,B 0,C 180,E1 -17650.197,E2 -17650.197} C_VEL
LIN {X 0,Y 286.279,Z 589.375,A -85,B 0,C 180,E1 -17651.721,E2 -17651.721} C_VEL
LIN {X 0,Y 283.686,Z 585.574,A -85,B 0,C 180,E1 -17652.656,E2 -17652.656} C_VEL
LIN {X 0,Y 280.949,Z 581.642,A -85,B 0,C 180,E1 -17653.707,E2 -17653.707} C_VEL
LIN {X 0,Y 278.445,Z 578.026,A -85,B 0,C 180,E1 -17654.748,E2 -17654.748} C_VEL
LIN {X 0,Y 275.356,Z 574.307,A -85,B 0,C 180,E1 -17656.094,E2 -17656.094} C_VEL
LIN {X 0,Y 274.5,Z 572.421,A -85,B 0,C 180,E1 -17656.568,E2 -17656.568} C_VEL
LIN {X 0,Y 271.98,Z 570.562,A -85,B 0,C 180,E1 -17657.727,E2 -17657.727} C_VEL
LIN {X 0,Y 270.576,Z 568.161,A -85,B 0,C 180,E1 -17658.553,E2 -17658.553} C_VEL
LIN {X 0,Y 270.295,Z 566.945,A -85,B 0,C 180,E1 -17658.868,E2 -17658.868} C_VEL
LIN {X 0,Y 270.213,Z 566.825,A -85,B 0,C 180,E1 -17661.354,E2 -17661.354} C_VEL
LIN {X 0,Y 270.266,Z 566.817,A -85,B 0,C 180,E1 -17664.586,E2 -17664.586} C_VEL
LIN {X 0,Y 270.264,Z 566.818,A -85,B 0,C 180,E1 -17667.909,E2 -17667.909} C_VEL
LIN {X 0,Y 270.238,Z 567.058,A -85,B 0,C 180,E1 -17670.263,E2 -17670.263} C_VEL
LIN {X 0,Y 271.321,Z 569.796,A -85,B 0,C 180,E1 -17674.741,E2 -17674.741} C_VEL
LIN {X 0,Y 272.508,Z 573.204,A -85,B 0,C 180,E1 -17678.24,E2 -17678.24} C_VEL
LIN {X 0,Y 273.683,Z 576.475,A -85,B 0,C 180,E1 -17680.906,E2 -17680.906} C_VEL
LIN {X 0,Y 275.066,Z 580.483,A -85,B 0,C 180,E1 -17683.619,E2 -17683.619} C_VEL
LIN {X 0,Y 276.735,Z 585.986,A -85,B 0,C 180,E1 -17686.712,E2 -17686.712} C_VEL
LIN {X 0,Y 278.616,Z 592.646,A -85,B 0,C 180,E1 -17689.889,E2 -17689.889} C_VEL
LIN {X 0,Y 280.338,Z 599.855,A -85,B 0,C 180,E1 -17692.771,E2 -17692.771} C_VEL
LIN {X 0,Y 283.315,Z 606.092,A -85,B 0,C 180,E1 -17693.984,E2 -17693.984} C_VEL
LIN {X 0,Y 287.062,Z 614.616,A -85,B 0,C 180,E1 -17695.402,E2 -17695.402} C_VEL
LIN {X 0,Y 289.52,Z 630.725,A -85,B 0,C 180,E1 -17696.835,E2 -17696.835} C_VEL
LIN {X 0,Y 291.599,Z 649.177,A -85,B 0,C 180,E1 -17698.204,E2 -17698.204} C_VEL
LIN {X 0,Y 292.692,Z 665.753,A -85,B 0,C 180,E1 -17699.227,E2 -17699.227} C_VEL
LIN {X 0,Y 293.155,Z 684.111,A -85,B 0,C 180,E1 -17700.156,E2 -17700.156} C_VEL
LIN {X 0,Y 290.679,Z 719.013,A -85,B 0,C 180,E1 -17701.38,E2 -17701.38} C_VEL
LIN {X 0,Y 288.923,Z 732.768,A -85,B 0,C 180,E1 -17702.081,E2 -17702.081} C_VEL
LIN {X 0,Y 286.624,Z 746.071,A -85,B 0,C 180,E1 -17703.026,E2 -17703.026} C_VEL
LIN {X 0,Y 283.706,Z 759.735,A -85,B 0,C 180,E1 -17704.311,E2 -17704.311} C_VEL
LIN {X 0,Y 281.907,Z 767.308,A -85,B 0,C 180,E1 -17705.172,E2 -17705.172} C_VEL
LIN {X 0,Y 280.485,Z 780.011,A -85,B 0,C 180,E1 -17706.073,E2 -17706.073} C_VEL
LIN {X 0,Y 278.893,Z 791.614,A -85,B 0,C 180,E1 -17707.206,E2 -17707.206} C_VEL
LIN {X 0,Y 277.123,Z 802.801,A -85,B 0,C 180,E1 -17708.621,E2 -17708.621} C_VEL
LIN {X 0,Y 275.257,Z 812.872,A -85,B 0,C 180,E1 -17710.228,E2 -17710.228} C_VEL
LIN {X 0,Y 273.655,Z 821.941,A -85,B 0,C 180,E1 -17712.052,E2 -17712.052} C_VEL
LIN {X 0,Y 272.115,Z 829.419,A -85,B 0,C 180,E1 -17713.882,E2 -17713.882} C_VEL
LIN {X 0,Y 270.653,Z 836.744,A -85,B 0,C 180,E1 -17716.104,E2 -17716.104} C_VEL
LIN {X 0,Y 269.71,Z 841.703,A -85,B 0,C 180,E1 -17717.969,E2 -17717.969} C_VEL
LIN {X 0,Y 268.978,Z 846.505,A -85,B 0,C 180,E1 -17720.223,E2 -17720.223} C_VEL
LIN {X 0,Y 268.492,Z 850.175,A -85,B 0,C 180,E1 -17722.481,E2 -17722.481} C_VEL
LIN {X 0,Y 268.268,Z 852.653,A -85,B 0,C 180,E1 -17724.571,E2 -17724.571} C_VEL
LIN {X 0,Y 268.256,Z 854.502,A -85,B 0,C 180,E1 -17726.998,E2 -17726.998} C_VEL
LIN {X 0,Y 268.27,Z 855.117,A -85,B 0,C 180,E1 -17728.5,E2 -17728.5} C_VEL
LIN {X 0,Y 268.299,Z 855.335,A -85,B 0,C 180,E1 -17730.001,E2 -17730.001} C_VEL
LIN {X 0,Y 268.26,Z 855.107,A -85,B 0,C 180,E1 -17731.502,E2 -17731.502} C_VEL
LIN {X 0,Y 268.251,Z 854.486,A -85,B 0,C 180,E1 -17733.005,E2 -17733.005} C_VEL
LIN {X 0,Y 268.326,Z 852.502,A -85,B 0,C 180,E1 -17735.558,E2 -17735.558} C_VEL
LIN {X 0,Y 268.636,Z 849.046,A -85,B 0,C 180,E1 -17738.274,E2 -17738.274} C_VEL
LIN {X 0,Y 269.197,Z 844.998,A -85,B 0,C 180,E1 -17740.531,E2 -17740.531} C_VEL
LIN {X 0,Y 270.174,Z 838.752,A -85,B 0,C 180,E1 -17743.158,E2 -17743.158} C_VEL
LIN {X 0,Y 271.628,Z 831.949,A -85,B 0,C 180,E1 -17745.38,E2 -17745.38} C_VEL
LIN {X 0,Y 272.991,Z 824.997,A -85,B 0,C 180,E1 -17747.222,E2 -17747.222} C_VEL
LIN {X 0,Y 274.491,Z 816.598,A -85,B 0,C 180,E1 -17749.054,E2 -17749.054} C_VEL
LIN {X 0,Y 276.396,Z 806.193,A -85,B 0,C 180,E1 -17750.855,E2 -17750.855} C_VEL
LIN {X 0,Y 278.43,Z 794.472,A -85,B 0,C 180,E1 -17752.445,E2 -17752.445} C_VEL
LIN {X 0,Y 280.101,Z 782.63,A -85,B 0,C 180,E1 -17753.67,E2 -17753.67} C_VEL
LIN {X 0,Y 281.538,Z 770.326,A -85,B 0,C 180,E1 -17754.619,E2 -17754.619} C_VEL
LIN {X 0,Y 282.709,Z 757.511,A -85,B 0,C 180,E1 -17755.295,E2 -17755.295} C_VEL
LIN {X 0,Y 283.426,Z 742.206,A -85,B 0,C 180,E1 -17755.768,E2 -17755.768} C_VEL
LIN {X 0,Y 284.893,Z 683.246,A -85,B 0,C 180,E1 -17757.244,E2 -17757.244} C_VEL
LIN {X 0,Y 282.082,Z 655.195,A -85,B 0,C 180,E1 -17758.325,E2 -17758.325} C_VEL
LIN {X 0,Y 279.373,Z 634.812,A -85,B 0,C 180,E1 -17759.222,E2 -17759.222} C_VEL
LIN {X 0,Y 278.126,Z 608.142,A -85,B 0,C 180,E1 -17761.844,E2 -17761.844} C_VEL
LIN {X 0,Y 277.52,Z 599.141,A -85,B 0,C 180,E1 -17762.724,E2 -17762.724} C_VEL
LIN {X 0,Y 275.78,Z 592.386,A -85,B 0,C 180,E1 -17763.642,E2 -17763.642} C_VEL
LIN {X 0,Y 272.968,Z 579.488,A -85,B 0,C 180,E1 -17767.458,E2 -17767.458} C_VEL
LIN {X 0,Y 270.21,Z 566.83,A -85,B 0,C 180,E1 -17771.401,E2 -17771.401} C_VEL
LIN {X 0,Y 270.169,Z 566.827,A -85,B 0,C 180,E1 -17775.383,E2 -17775.383} C_VEL
LIN {X 0,Y 270.176,Z 566.821,A -85,B 0,C 180,E1 -17779.434,E2 -17779.434} C_VEL
LIN {X 0,Y 270.227,Z 566.808,A -85,B 0,C 180,E1 -17783.731,E2 -17783.731} C_VEL
LIN {X 0,Y 270.205,Z 566.824,A -85,B 0,C 180,E1 -17786.893,E2 -17786.893} C_VEL
LIN {X 0,Y 270.231,Z 566.813,A -85,B 0,C 180,E1 -17790.387,E2 -17790.387} C_VEL
LIN {X 0,Y 270.264,Z 566.808,A -85,B 0,C 180,E1 -17793.764,E2 -17793.764} C_VEL
LIN {X 0,Y 270.212,Z 566.816,A -85,B 0,C 180,E1 -17797.037,E2 -17797.037} C_VEL
LIN {X 0,Y 270.303,Z 566.806,A -85,B 0,C 180,E1 -17800.245,E2 -17800.245} C_VEL
LIN {X 0,Y 270.399,Z 566.799,A -85,B 0,C 180,E1 -17804.935,E2 -17804.935} C_VEL
LIN {X 0,Y 270.415,Z 566.772,A -85,B 0,C 180,E1 -17809.518,E2 -17809.518} C_VEL
LIN {X 0,Y 270.601,Z 566.776,A -85,B 0,C 180,E1 -17812.539,E2 -17812.539} C_VEL
LIN {X 0,Y 270.788,Z 566.731,A -85,B 0,C 180,E1 -17818.513,E2 -17818.513} C_VEL
LIN {X 0,Y 270.789,Z 566.756,A -85,B 0,C 180,E1 -17821.487,E2 -17821.487} C_VEL
LIN {X 0,Y 270.61,Z 566.769,A -85,B 0,C 180,E1 -17827.461,E2 -17827.461} C_VEL
LIN {X 0,Y 270.444,Z 566.788,A -85,B 0,C 180,E1 -17830.481,E2 -17830.481} C_VEL
LIN {X 0,Y 270.399,Z 566.8,A -85,B 0,C 180,E1 -17835.065,E2 -17835.065} C_VEL
LIN {X 0,Y 270.304,Z 566.792,A -85,B 0,C 180,E1 -17839.756,E2 -17839.756} C_VEL
LIN {X 0,Y 270.276,Z 566.801,A -85,B 0,C 180,E1 -17844.586,E2 -17844.586} C_VEL
LIN {X 0,Y 270.274,Z 566.819,A -85,B 0,C 180,E1 -17847.909,E2 -17847.909} C_VEL
LIN {X 0,Y 270.187,Z 566.815,A -85,B 0,C 180,E1 -17851.348,E2 -17851.348} C_VEL
LIN {X 0,Y 270.206,Z 566.818,A -85,B 0,C 180,E1 -17854.905,E2 -17854.905} C_VEL
LIN {X 0,Y 270.225,Z 566.822,A -85,B 0,C 180,E1 -17858.717,E2 -17858.717} C_VEL
LIN {X 0,Y 270.168,Z 566.824,A -85,B 0,C 180,E1 -17863.249,E2 -17863.249} C_VEL
LIN {X 0,Y 270.174,Z 566.851,A -85,B 0,C 180,E1 -17866.687,E2 -17866.687} C_VEL
LIN {X 0,Y 274.418,Z 579.084,A -85,B 0,C 180,E1 -17870.204,E2 -17870.204} C_VEL
LIN {X 0,Y 277.473,Z 589.108,A -85,B 0,C 180,E1 -17872.924,E2 -17872.924} C_VEL
LIN {X 0,Y 280.636,Z 601.731,A -85,B 0,C 180,E1 -17876.071,E2 -17876.071} C_VEL
LIN {X 0,Y 282.417,Z 610.299,A -85,B 0,C 180,E1 -17878.087,E2 -17878.087} C_VEL
LIN {X 0,Y 281.559,Z 619.66,A -85,B 0,C 180,E1 -17879.844,E2 -17879.844} C_VEL
LIN {X 0,Y 280.979,Z 625.414,A -85,B 0,C 180,E1 -17880.884,E2 -17880.884} C_VEL
LIN {X 0,Y 285.445,Z 653.292,A -85,B 0,C 180,E1 -17882.172,E2 -17882.172} C_VEL
LIN {X 0,Y 286.219,Z 659.56,A -85,B 0,C 180,E1 -17882.429,E2 -17882.429} C_VEL
LIN {X 0,Y 283.815,Z 738.263,A -85,B 0,C 180,E1 -17884.417,E2 -17884.417} C_VEL
LIN {X 0,Y 282.914,Z 751.32,A -85,B 0,C 180,E1 -17885.019,E2 -17885.019} C_VEL
LIN {X 0,Y 281.542,Z 764.848,A -85,B 0,C 180,E1 -17885.97,E2 -17885.97} C_VEL
LIN {X 0,Y 280.03,Z 776.595,A -85,B 0,C 180,E1 -17887.106,E2 -17887.106} C_VEL
LIN {X 0,Y 278.23,Z 787.792,A -85,B 0,C 180,E1 -17888.514,E2 -17888.514} C_VEL
LIN {X 0,Y 276.525,Z 797.847,A -85,B 0,C 180,E1 -17890.115,E2 -17890.115} C_VEL
LIN {X 0,Y 275.049,Z 806.2,A -85,B 0,C 180,E1 -17891.758,E2 -17891.758} C_VEL
LIN {X 0,Y 273.088,Z 815.182,A -85,B 0,C 180,E1 -17893.938,E2 -17893.938} C_VEL
LIN {X 0,Y 271.6,Z 822.391,A -85,B 0,C 180,E1 -17896.15,E2 -17896.15} C_VEL
LIN {X 0,Y 270.171,Z 829.007,A -85,B 0,C 180,E1 -17898.748,E2 -17898.748} C_VEL
LIN {X 0,Y 269.331,Z 833.345,A -85,B 0,C 180,E1 -17900.991,E2 -17900.991} C_VEL
LIN {X 0,Y 268.711,Z 837.092,A -85,B 0,C 180,E1 -17903.655,E2 -17903.655} C_VEL
LIN {X 0,Y 268.469,Z 838.902,A -85,B 0,C 180,E1 -17905.495,E2 -17905.495} C_VEL
LIN {X 0,Y 268.33,Z 839.897,A -85,B 0,C 180,E1 -17906.996,E2 -17906.996} C_VEL
LIN {X 0,Y 268.208,Z 840.743,A -85,B 0,C 180,E1 -17909.999,E2 -17909.999} C_VEL
LIN {X 0,Y 268.229,Z 840.548,A -85,B 0,C 180,E1 -17911.5,E2 -17911.5} C_VEL
LIN {X 0,Y 268.326,Z 839.96,A -85,B 0,C 180,E1 -17913.001,E2 -17913.001} C_VEL
LIN {X 0,Y 268.466,Z 838.991,A -85,B 0,C 180,E1 -17914.503,E2 -17914.503} C_VEL
LIN {X 0,Y 268.71,Z 837.232,A -85,B 0,C 180,E1 -17916.343,E2 -17916.343} C_VEL
LIN {X 0,Y 269.295,Z 833.539,A -85,B 0,C 180,E1 -17919.007,E2 -17919.007} C_VEL
LIN {X 0,Y 270.139,Z 829.258,A -85,B 0,C 180,E1 -17921.25,E2 -17921.25} C_VEL
LIN {X 0,Y 271.299,Z 823.791,A -85,B 0,C 180,E1 -17923.481,E2 -17923.481} C_VEL
LIN {X 0,Y 272.719,Z 816.93,A -85,B 0,C 180,E1 -17925.698,E2 -17925.698} C_VEL
LIN {X 0,Y 274.616,Z 808.327,A -85,B 0,C 180,E1 -17927.883,E2 -17927.883} C_VEL
LIN {X 0,Y 276.397,Z 798.903,A -85,B 0,C 180,E1 -17929.812,E2 -17929.812} C_VEL
LIN {X 0,Y 278.169,Z 788.573,A -85,B 0,C 180,E1 -17931.489,E2 -17931.489} C_VEL
LIN {X 0,Y 279.962,Z 777.549,A -85,B 0,C 180,E1 -17932.897,E2 -17932.897} C_VEL
LIN {X 0,Y 281.496,Z 766.158,A -85,B 0,C 180,E1 -17934.032,E2 -17934.032} C_VEL
LIN {X 0,Y 282.78,Z 753.097,A -85,B 0,C 180,E1 -17934.991,E2 -17934.991} C_VEL
LIN {X 0,Y 283.748,Z 740.074,A -85,B 0,C 180,E1 -17935.636,E2 -17935.636} C_VEL
LIN {X 0,Y 284.563,Z 717.72,A -85,B 0,C 180,E1 -17936.245,E2 -17936.245} C_VEL
LIN {X 0,Y 286.163,Z 661.399,A -85,B 0,C 180,E1 -17937.646,E2 -17937.646} C_VEL
LIN {X 0,Y 281.963,Z 636.423,A -85,B 0,C 180,E1 -17938.807,E2 -17938.807} C_VEL
LIN {X 0,Y 280.049,Z 626.193,A -85,B 0,C 180,E1 -17939.347,E2 -17939.347} C_VEL
LIN {X 0,Y 281.656,Z 611.176,A -85,B 0,C 180,E1 -17942.441,E2 -17942.441} C_VEL
LIN {X 0,Y 281.27,Z 607.436,A -85,B 0,C 180,E1 -17943.345,E2 -17943.345} C_VEL
LIN {X 0,Y 278.98,Z 596.345,A -85,B 0,C 180,E1 -17946.28,E2 -17946.28} C_VEL
LIN {X 0,Y 276.035,Z 584.955,A -85,B 0,C 180,E1 -17949.53,E2 -17949.53} C_VEL
LIN {X 0,Y 272.633,Z 573.804,A -85,B 0,C 180,E1 -17952.988,E2 -17952.988} C_VEL
LIN {X 0,Y 279.593,Z 592.87,A -85,B 0,C 180,E1 -17954.102,E2 -17954.102} C_VEL
LIN {X 0,Y 278.211,Z 641.235,A -85,B 0,C 180,E1 -17955.682,E2 -17955.682} C_VEL
LIN {X 0,Y 277.989,Z 655.601,A -85,B 0,C 180,E1 -17956.298,E2 -17956.298} C_VEL
LIN {X 0,Y 277.627,Z 665.676,A -85,B 0,C 180,E1 -17956.921,E2 -17956.921} C_VEL
LIN {X 0,Y 276.683,Z 671.269,A -85,B 0,C 180,E1 -17957.308,E2 -17957.308} C_VEL
LIN {X 0,Y 273.363,Z 680.103,A -85,B 0,C 180,E1 -17957.948,E2 -17957.948} C_VEL
LIN {X 0,Y 269.957,Z 688.656,A -85,B 0,C 180,E1 -17958.719,E2 -17958.719} C_VEL
LIN {X 0,Y 268.943,Z 693.723,A -85,B 0,C 180,E1 -17959.313,E2 -17959.313} C_VEL
LIN {X 0,Y 267.871,Z 705.256,A -85,B 0,C 180,E1 -17960.974,E2 -17960.974} C_VEL
LIN {X 0,Y 266.8,Z 716.12,A -85,B 0,C 180,E1 -17962.946,E2 -17962.946} C_VEL
LIN {X 0,Y 265.821,Z 725.505,A -85,B 0,C 180,E1 -17965.042,E2 -17965.042} C_VEL
LIN {X 0,Y 264.836,Z 734.255,A -85,B 0,C 180,E1 -17967.494,E2 -17967.494} C_VEL
LIN {X 0,Y 264.303,Z 740.445,A -85,B 0,C 180,E1 -17969.654,E2 -17969.654} C_VEL
LIN {X 0,Y 263.821,Z 746.386,A -85,B 0,C 180,E1 -17972.272,E2 -17972.272} C_VEL
LIN {X 0,Y 263.596,Z 750.961,A -85,B 0,C 180,E1 -17975.022,E2 -17975.022} C_VEL
LIN {X 0,Y 263.581,Z 752.742,A -85,B 0,C 180,E1 -17976.425,E2 -17976.425} C_VEL
LIN {X 0,Y 263.825,Z 754.91,A -85,B 0,C 180,E1 -17978.8,E2 -17978.8} C_VEL
LIN {X 0,Y 264.427,Z 756.129,A -85,B 0,C 180,E1 -17981.401,E2 -17981.401} C_VEL
LIN {X 0,Y 264.928,Z 756.242,A -85,B 0,C 180,E1 -17983.034,E2 -17983.034} C_VEL
LIN {X 0,Y 265.592,Z 755.898,A -85,B 0,C 180,E1 -17984.656,E2 -17984.656} C_VEL
LIN {X 0,Y 266.794,Z 754.491,A -85,B 0,C 180,E1 -17987.067,E2 -17987.067} C_VEL
LIN {X 0,Y 268.809,Z 750.939,A -85,B 0,C 180,E1 -17990.215,E2 -17990.215} C_VEL
LIN {X 0,Y 270.731,Z 746.91,A -85,B 0,C 180,E1 -17992.542,E2 -17992.542} C_VEL
LIN {X 0,Y 272.855,Z 741.646,A -85,B 0,C 180,E1 -17994.828,E2 -17994.828} C_VEL
LIN {X 0,Y 275.296,Z 734.881,A -85,B 0,C 180,E1 -17997.073,E2 -17997.073} C_VEL
LIN {X 0,Y 278.025,Z 726.43,A -85,B 0,C 180,E1 -17999.276,E2 -17999.276} C_VEL
LIN {X 0,Y 280.341,Z 717.82,A -85,B 0,C 180,E1 -18001.077,E2 -18001.077} C_VEL
LIN {X 0,Y 282.932,Z 707.001,A -85,B 0,C 180,E1 -18002.848,E2 -18002.848} C_VEL
LIN {X 0,Y 285.011,Z 696.404,A -85,B 0,C 180,E1 -18004.242,E2 -18004.242} C_VEL
LIN {X 0,Y 286.814,Z 684.789,A -85,B 0,C 180,E1 -18005.448,E2 -18005.448} C_VEL
LIN {X 0,Y 288.302,Z 671.883,A -85,B 0,C 180,E1 -18006.474,E2 -18006.474} C_VEL
LIN {X 0,Y 289.151,Z 658.733,A -85,B 0,C 180,E1 -18007.226,E2 -18007.226} C_VEL
LIN {X 0,Y 290.658,Z 631.067,A -85,B 0,C 180,E1 -18008.342,E2 -18008.342} C_VEL
LIN {X 0,Y 292.21,Z 611.709,A -85,B 0,C 180,E1 -18009.049,E2 -18009.049} C_VEL
LIN {X 0,Y 286.772,Z 601.23,A -85,B 0,C 180,E1 -18010.869,E2 -18010.869} C_VEL
LIN {X 0,Y 282.524,Z 594.435,A -85,B 0,C 180,E1 -18012.404,E2 -18012.404} C_VEL
LIN {X 0,Y 280.268,Z 591.107,A -85,B 0,C 180,E1 -18013.258,E2 -18013.258} C_VEL
LIN {X 0,Y 277.914,Z 587.552,A -85,B 0,C 180,E1 -18014.24,E2 -18014.24} C_VEL
LIN {X 0,Y 274.91,Z 583.286,A -85,B 0,C 180,E1 -18015.541,E2 -18015.541} C_VEL
LIN {X 0,Y 272.5,Z 580.153,A -85,B 0,C 180,E1 -18016.693,E2 -18016.693} C_VEL
LIN {X 0,Y 271.858,Z 578.818,A -85,B 0,C 180,E1 -18017.053,E2 -18017.053} C_VEL
LIN {X 0,Y 269.255,Z 576.497,A -85,B 0,C 180,E1 -18018.352,E2 -18018.352} C_VEL
LIN {X 0,Y 267.562,Z 573.341,A -85,B 0,C 180,E1 -18019.457,E2 -18019.457} C_VEL
LIN {X 0,Y 264.864,Z 571.442,A -85,B 0,C 180,E1 -18021.095,E2 -18021.095} C_VEL
LIN {X 0,Y 263.894,Z 570.087,A -85,B 0,C 180,E1 -18021.891,E2 -18021.891} C_VEL
LIN {X 0,Y 263.859,Z 569.912,A -85,B 0,C 180,E1 -18025.225,E2 -18025.225} C_VEL
LIN {X 0,Y 264.159,Z 570.496,A -85,B 0,C 180,E1 -18028.613,E2 -18028.613} C_VEL
LIN {X 0,Y 264.548,Z 571.952,A -85,B 0,C 180,E1 -18031.78,E2 -18031.78} C_VEL
LIN {X 0,Y 265.483,Z 573.92,A -85,B 0,C 180,E1 -18034.854,E2 -18034.854} C_VEL
LIN {X 0,Y 266.362,Z 576.546,A -85,B 0,C 180,E1 -18037.672,E2 -18037.672} C_VEL
LIN {X 0,Y 267.775,Z 580.524,A -85,B 0,C 180,E1 -18041.007,E2 -18041.007} C_VEL
LIN {X 0,Y 269.137,Z 584.595,A -85,B 0,C 180,E1 -18043.788,E2 -18043.788} C_VEL
LIN {X 0,Y 270.63,Z 589.61,A -85,B 0,C 180,E1 -18046.647,E2 -18046.647} C_VEL
LIN {X 0,Y 272.521,Z 596.645,A -85,B 0,C 180,E1 -18050.061,E2 -18050.061} C_VEL
LIN {X 0,Y 276.066,Z 603.826,A -85,B 0,C 180,E1 -18051.77,E2 -18051.77} C_VEL
LIN {X 0,Y 277.202,Z 606.174,A -85,B 0,C 180,E1 -18052.28,E2 -18052.28} C_VEL
LIN {X 0,Y 280.41,Z 613.038,A -85,B 0,C 180,E1 -18053.634,E2 -18053.634} C_VEL
LIN {X 0,Y 282.763,Z 618.692,A -85,B 0,C 180,E1 -18054.594,E2 -18054.594} C_VEL
LIN {X 0,Y 285.103,Z 635.975,A -85,B 0,C 180,E1 -18056.144,E2 -18056.144} C_VEL
LIN {X 0,Y 286.781,Z 653.512,A -85,B 0,C 180,E1 -18057.449,E2 -18057.449} C_VEL
LIN {X 0,Y 287.65,Z 670.404,A -85,B 0,C 180,E1 -18058.494,E2 -18058.494} C_VEL
LIN {X 0,Y 287.721,Z 686.637,A -85,B 0,C 180,E1 -18059.316,E2 -18059.316} C_VEL
LIN {X 0,Y 285.291,Z 718.216,A -85,B 0,C 180,E1 -18060.441,E2 -18060.441} C_VEL
LIN {X 0,Y 283.398,Z 732.346,A -85,B 0,C 180,E1 -18061.184,E2 -18061.184} C_VEL
LIN {X 0,Y 280.782,Z 746.296,A -85,B 0,C 180,E1 -18062.215,E2 -18062.215} C_VEL
LIN {X 0,Y 278.116,Z 758.021,A -85,B 0,C 180,E1 -18063.352,E2 -18063.352} C_VEL
LIN {X 0,Y 275.271,Z 769.316,A -85,B 0,C 180,E1 -18064.683,E2 -18064.683} C_VEL
LIN {X 0,Y 273.884,Z 780.826,A -85,B 0,C 180,E1 -18065.56,E2 -18065.56} C_VEL
LIN {X 0,Y 272.119,Z 793.005,A -85,B 0,C 180,E1 -18066.807,E2 -18066.807} C_VEL
LIN {X 0,Y 270.266,Z 803.871,A -85,B 0,C 180,E1 -18068.252,E2 -18068.252} C_VEL
LIN {X 0,Y 268.161,Z 814.627,A -85,B 0,C 180,E1 -18070.082,E2 -18070.082} C_VEL
LIN {X 0,Y 266.54,Z 823.376,A -85,B 0,C 180,E1 -18071.953,E2 -18071.953} C_VEL
LIN {X 0,Y 265.041,Z 830.581,A -85,B 0,C 180,E1 -18073.835,E2 -18073.835} C_VEL
LIN {X 0,Y 263.503,Z 837.64,A -85,B 0,C 180,E1 -18076.112,E2 -18076.112} C_VEL
LIN {X 0,Y 262.442,Z 843.255,A -85,B 0,C 180,E1 -18078.415,E2 -18078.415} C_VEL
LIN {X 0,Y 261.742,Z 847.661,A -85,B 0,C 180,E1 -18080.73,E2 -18080.73} C_VEL
LIN {X 0,Y 261.418,Z 849.982,A -85,B 0,C 180,E1 -18082.276,E2 -18082.276} C_VEL
LIN {X 0,Y 261.184,Z 852.652,A -85,B 0,C 180,E1 -18084.627,E2 -18084.627} C_VEL
LIN {X 0,Y 261.168,Z 854.309,A -85,B 0,C 180,E1 -18086.916,E2 -18086.916} C_VEL
LIN {X 0,Y 261.194,Z 854.925,A -85,B 0,C 180,E1 -18088.459,E2 -18088.459} C_VEL
LIN {X 0,Y 261.221,Z 855.142,A -85,B 0,C 180,E1 -18090.001,E2 -18090.001} C_VEL
LIN {X 0,Y 261.185,Z 854.915,A -85,B 0,C 180,E1 -18091.543,E2 -18091.543} C_VEL
LIN {X 0,Y 261.163,Z 854.292,A -85,B 0,C 180,E1 -18093.086,E2 -18093.086} C_VEL
LIN {X 0,Y 261.221,Z 852.544,A -85,B 0,C 180,E1 -18095.459,E2 -18095.459} C_VEL
LIN {X 0,Y 261.582,Z 848.852,A -85,B 0,C 180,E1 -18098.499,E2 -18098.499} C_VEL
LIN {X 0,Y 262.167,Z 844.803,A -85,B 0,C 180,E1 -18100.817,E2 -18100.817} C_VEL
LIN {X 0,Y 263.232,Z 838.559,A -85,B 0,C 180,E1 -18103.511,E2 -18103.511} C_VEL
LIN {X 0,Y 264.768,Z 831.757,A -85,B 0,C 180,E1 -18105.789,E2 -18105.789} C_VEL
LIN {X 0,Y 266.191,Z 824.845,A -85,B 0,C 180,E1 -18107.666,E2 -18107.666} C_VEL
LIN {X 0,Y 267.759,Z 816.408,A -85,B 0,C 180,E1 -18109.552,E2 -18109.552} C_VEL
LIN {X 0,Y 269.772,Z 806.007,A -85,B 0,C 180,E1 -18111.391,E2 -18111.391} C_VEL
LIN {X 0,Y 271.893,Z 794.289,A -85,B 0,C 180,E1 -18113.015,E2 -18113.015} C_VEL
LIN {X 0,Y 273.601,Z 782.452,A -85,B 0,C 180,E1 -18114.268,E2 -18114.268} C_VEL
LIN {X 0,Y 275.082,Z 770.157,A -85,B 0,C 180,E1 -18115.237,E2 -18115.237} C_VEL
LIN {X 0,Y 276.325,Z 757.367,A -85,B 0,C 180,E1 -18115.923,E2 -18115.923} C_VEL
LIN {X 0,Y 277.058,Z 742.106,A -85,B 0,C 180,E1 -18116.405,E2 -18116.405} C_VEL
LIN {X 0,Y 278.585,Z 683.931,A -85,B 0,C 180,E1 -18117.892,E2 -18117.892} C_VEL
LIN {X 0,Y 275.934,Z 656.888,A -85,B 0,C 180,E1 -18118.963,E2 -18118.963} C_VEL
LIN {X 0,Y 273.024,Z 634.643,A -85,B 0,C 180,E1 -18119.971,E2 -18119.971} C_VEL
LIN {X 0,Y 271.952,Z 608.493,A -85,B 0,C 180,E1 -18122.648,E2 -18122.648} C_VEL
LIN {X 0,Y 271.505,Z 601.207,A -85,B 0,C 180,E1 -18123.405,E2 -18123.405} C_VEL
LIN {X 0,Y 269.825,Z 595.337,A -85,B 0,C 180,E1 -18124.211,E2 -18124.211} C_VEL
LIN {X 0,Y 267.69,Z 588.377,A -85,B 0,C 180,E1 -18125.282,E2 -18125.282} C_VEL
LIN {X 0,Y 264.64,Z 574.365,A -85,B 0,C 180,E1 -18129.633,E2 -18129.633} C_VEL
LIN {X 0,Y 263.156,Z 567.706,A -85,B 0,C 180,E1 -18131.809,E2 -18131.809} C_VEL
LIN {X 0,Y 263.132,Z 567.709,A -85,B 0,C 180,E1 -18136.15,E2 -18136.15} C_VEL
LIN {X 0,Y 263.108,Z 567.71,A -85,B 0,C 180,E1 -18140.128,E2 -18140.128} C_VEL
LIN {X 0,Y 263.164,Z 567.688,A -85,B 0,C 180,E1 -18144.018,E2 -18144.018} C_VEL
LIN {X 0,Y 263.135,Z 567.694,A -85,B 0,C 180,E1 -18147.712,E2 -18147.712} C_VEL
LIN {X 0,Y 263.204,Z 567.7,A -85,B 0,C 180,E1 -18151.783,E2 -18151.783} C_VEL
LIN {X 0,Y 263.203,Z 567.675,A -85,B 0,C 180,E1 -18155.212,E2 -18155.212} C_VEL
LIN {X 0,Y 263.265,Z 567.686,A -85,B 0,C 180,E1 -18159.694,E2 -18159.694} C_VEL
LIN {X 0,Y 263.347,Z 567.676,A -85,B 0,C 180,E1 -18164.522,E2 -18164.522} C_VEL
LIN {X 0,Y 263.357,Z 567.651,A -85,B 0,C 180,E1 -18169.234,E2 -18169.234} C_VEL
LIN {X 0,Y 263.56,Z 567.652,A -85,B 0,C 180,E1 -18172.338,E2 -18172.338} C_VEL
LIN {X 0,Y 263.752,Z 567.606,A -85,B 0,C 180,E1 -18178.473,E2 -18178.473} C_VEL
LIN {X 0,Y 263.753,Z 567.632,A -85,B 0,C 180,E1 -18181.527,E2 -18181.527} C_VEL
LIN {X 0,Y 263.572,Z 567.647,A -85,B 0,C 180,E1 -18187.662,E2 -18187.662} C_VEL
LIN {X 0,Y 263.376,Z 567.663,A -85,B 0,C 180,E1 -18190.766,E2 -18190.766} C_VEL
LIN {X 0,Y 263.347,Z 567.68,A -85,B 0,C 180,E1 -18195.478,E2 -18195.478} C_VEL
LIN {X 0,Y 263.266,Z 567.672,A -85,B 0,C 180,E1 -18200.307,E2 -18200.307} C_VEL
LIN {X 0,Y 263.21,Z 567.678,A -85,B 0,C 180,E1 -18205.291,E2 -18205.291} C_VEL
LIN {X 0,Y 263.182,Z 567.701,A -85,B 0,C 180,E1 -18208.73,E2 -18208.73} C_VEL
LIN {X 0,Y 263.135,Z 567.703,A -85,B 0,C 180,E1 -18212.288,E2 -18212.288} C_VEL
LIN {X 0,Y 263.2,Z 567.697,A -85,B 0,C 180,E1 -18216.767,E2 -18216.767} C_VEL
LIN {X 0,Y 263.118,Z 567.702,A -85,B 0,C 180,E1 -18219.871,E2 -18219.871} C_VEL
LIN {X 0,Y 263.106,Z 567.706,A -85,B 0,C 180,E1 -18223.988,E2 -18223.988} C_VEL
LIN {X 0,Y 263.119,Z 567.765,A -85,B 0,C 180,E1 -18225.603,E2 -18225.603} C_VEL
LIN {X 0,Y 267.785,Z 580.908,A -85,B 0,C 180,E1 -18229.562,E2 -18229.562} C_VEL
LIN {X 0,Y 271.192,Z 592.078,A -85,B 0,C 180,E1 -18232.63,E2 -18232.63} C_VEL
LIN {X 0,Y 274.351,Z 604.988,A -85,B 0,C 180,E1 -18235.918,E2 -18235.918} C_VEL
LIN {X 0,Y 275.961,Z 613.031,A -85,B 0,C 180,E1 -18237.804,E2 -18237.804} C_VEL
LIN {X 0,Y 274.644,Z 625.575,A -85,B 0,C 180,E1 -18240.142,E2 -18240.142} C_VEL
LIN {X 0,Y 279.19,Z 654.116,A -85,B 0,C 180,E1 -18241.513,E2 -18241.513} C_VEL
LIN {X 0,Y 279.937,Z 660.13,A -85,B 0,C 180,E1 -18241.769,E2 -18241.769} C_VEL
LIN {X 0,Y 277.431,Z 738.396,A -85,B 0,C 180,E1 -18243.784,E2 -18243.784} C_VEL
LIN {X 0,Y 276.517,Z 751.483,A -85,B 0,C 180,E1 -18244.4,E2 -18244.4} C_VEL
LIN {X 0,Y 275.221,Z 763.947,A -85,B 0,C 180,E1 -18245.281,E2 -18245.281} C_VEL
LIN {X 0,Y 273.76,Z 775.146,A -85,B 0,C 180,E1 -18246.35,E2 -18246.35} C_VEL
LIN {X 0,Y 271.857,Z 786.727,A -85,B 0,C 180,E1 -18247.784,E2 -18247.784} C_VEL
LIN {X 0,Y 270.068,Z 796.908,A -85,B 0,C 180,E1 -18249.402,E2 -18249.402} C_VEL
LIN {X 0,Y 268.317,Z 806.39,A -85,B 0,C 180,E1 -18251.284,E2 -18251.284} C_VEL
LIN {X 0,Y 266.281,Z 815.373,A -85,B 0,C 180,E1 -18253.516,E2 -18253.516} C_VEL
LIN {X 0,Y 264.706,Z 822.583,A -85,B 0,C 180,E1 -18255.782,E2 -18255.782} C_VEL
LIN {X 0,Y 263.217,Z 829.2,A -85,B 0,C 180,E1 -18258.447,E2 -18258.447} C_VEL
LIN {X 0,Y 262.313,Z 833.538,A -85,B 0,C 180,E1 -18260.748,E2 -18260.748} C_VEL
LIN {X 0,Y 261.63,Z 837.501,A -85,B 0,C 180,E1 -18263.674,E2 -18263.674} C_VEL
LIN {X 0,Y 261.383,Z 839.096,A -85,B 0,C 180,E1 -18265.372,E2 -18265.372} C_VEL
LIN {X 0,Y 261.246,Z 840.09,A -85,B 0,C 180,E1 -18266.915,E2 -18266.915} C_VEL
LIN {X 0,Y 261.16,Z 840.703,A -85,B 0,C 180,E1 -18268.457,E2 -18268.457} C_VEL
LIN {X 0,Y 261.134,Z 840.935,A -85,B 0,C 180,E1 -18269.999,E2 -18269.999} C_VEL
LIN {X 0,Y 261.158,Z 840.74,A -85,B 0,C 180,E1 -18271.541,E2 -18271.541} C_VEL
LIN {X 0,Y 261.243,Z 840.152,A -85,B 0,C 180,E1 -18273.083,E2 -18273.083} C_VEL
LIN {X 0,Y 261.38,Z 839.183,A -85,B 0,C 180,E1 -18274.625,E2 -18274.625} C_VEL
LIN {X 0,Y 261.629,Z 837.64,A -85,B 0,C 180,E1 -18276.324,E2 -18276.324} C_VEL
LIN {X 0,Y 262.286,Z 833.73,A -85,B 0,C 180,E1 -18279.25,E2 -18279.25} C_VEL
LIN {X 0,Y 263.186,Z 829.448,A -85,B 0,C 180,E1 -18281.552,E2 -18281.552} C_VEL
LIN {X 0,Y 264.403,Z 823.98,A -85,B 0,C 180,E1 -18283.839,E2 -18283.839} C_VEL
LIN {X 0,Y 265.893,Z 817.117,A -85,B 0,C 180,E1 -18286.111,E2 -18286.111} C_VEL
LIN {X 0,Y 267.863,Z 808.512,A -85,B 0,C 180,E1 -18288.35,E2 -18288.35} C_VEL
LIN {X 0,Y 269.638,Z 799.578,A -85,B 0,C 180,E1 -18290.227,E2 -18290.227} C_VEL
LIN {X 0,Y 271.376,Z 789.998,A -85,B 0,C 180,E1 -18291.855,E2 -18291.855} C_VEL
LIN {X 0,Y 273.215,Z 779.246,A -85,B 0,C 180,E1 -18293.295,E2 -18293.295} C_VEL
LIN {X 0,Y 274.915,Z 767.281,A -85,B 0,C 180,E1 -18294.544,E2 -18294.544} C_VEL
LIN {X 0,Y 276.269,Z 754.667,A -85,B 0,C 180,E1 -18295.521,E2 -18295.521} C_VEL
LIN {X 0,Y 277.303,Z 741.224,A -85,B 0,C 180,E1 -18296.226,E2 -18296.226} C_VEL
LIN {X 0,Y 277.959,Z 724.897,A -85,B 0,C 180,E1 -18296.715,E2 -18296.715} C_VEL
LIN {X 0,Y 279.839,Z 661.986,A -85,B 0,C 180,E1 -18298.312,E2 -18298.312} C_VEL
LIN {X 0,Y 275.766,Z 637.62,A -85,B 0,C 180,E1 -18299.484,E2 -18299.484} C_VEL
LIN {X 0,Y 273.661,Z 626.294,A -85,B 0,C 180,E1 -18300.097,E2 -18300.097} C_VEL
LIN {X 0,Y 275.138,Z 613.105,A -85,B 0,C 180,E1 -18302.872,E2 -18302.872} C_VEL
LIN {X 0,Y 274.298,Z 607.363,A -85,B 0,C 180,E1 -18304.308,E2 -18304.308} C_VEL
LIN {X 0,Y 271.882,Z 596.292,A -85,B 0,C 180,E1 -18307.357,E2 -18307.357} C_VEL
LIN {X 0,Y 268.87,Z 584.941,A -85,B 0,C 180,E1 -18310.709,E2 -18310.709} C_VEL
LIN {X 0,Y 266.885,Z 578.425,A -85,B 0,C 180,E1 -18312.782,E2 -18312.782} C_VEL
LIN {X 0,Y 272.667,Z 594.14,A -85,B 0,C 180,E1 -18313.726,E2 -18313.726} C_VEL
LIN {X 0,Y 271.28,Z 645.822,A -85,B 0,C 180,E1 -18315.49,E2 -18315.49} C_VEL
LIN {X 0,Y 271.016,Z 659.505,A -85,B 0,C 180,E1 -18316.158,E2 -18316.158} C_VEL
LIN {X 0,Y 270.372,Z 672.968,A -85,B 0,C 180,E1 -18317.124,E2 -18317.124} C_VEL
LIN {X 0,Y 269.557,Z 685.508,A -85,B 0,C 180,E1 -18318.329,E2 -18318.329} C_VEL
LIN {X 0,Y 268.943,Z 693.723,A -85,B 0,C 180,E1 -18319.313,E2 -18319.313} C_VEL
LIN {X 0,Y 267.914,Z 698.705,A -85,B 0,C 180,E1 -18319.953,E2 -18319.953} C_VEL
LIN {X 0,Y 264.381,Z 706.556,A -85,B 0,C 180,E1 -18321.013,E2 -18321.013} C_VEL
LIN {X 0,Y 260.761,Z 714.031,A -85,B 0,C 180,E1 -18322.211,E2 -18322.211} C_VEL
LIN {X 0,Y 259.619,Z 718.369,A -85,B 0,C 180,E1 -18323.056,E2 -18323.056} C_VEL
LIN {X 0,Y 258.634,Z 727.46,A -85,B 0,C 180,E1 -18325.205,E2 -18325.205} C_VEL
LIN {X 0,Y 257.716,Z 735.987,A -85,B 0,C 180,E1 -18327.709,E2 -18327.709} C_VEL
LIN {X 0,Y 257.151,Z 742.439,A -85,B 0,C 180,E1 -18330.081,E2 -18330.081} C_VEL
LIN {X 0,Y 256.753,Z 747.204,A -85,B 0,C 180,E1 -18332.268,E2 -18332.268} C_VEL
LIN {X 0,Y 256.555,Z 751.304,A -85,B 0,C 180,E1 -18334.683,E2 -18334.683} C_VEL
LIN {X 0,Y 256.609,Z 754.647,A -85,B 0,C 180,E1 -18337.453,E2 -18337.453} C_VEL
LIN {X 0,Y 256.854,Z 756.065,A -85,B 0,C 180,E1 -18339.163,E2 -18339.163} C_VEL
LIN {X 0,Y 257.255,Z 756.954,A -85,B 0,C 180,E1 -18340.863,E2 -18340.863} C_VEL
LIN {X 0,Y 257.753,Z 757.365,A -85,B 0,C 180,E1 -18342.609,E2 -18342.609} C_VEL
LIN {X 0,Y 258.393,Z 757.305,A -85,B 0,C 180,E1 -18344.217,E2 -18344.217} C_VEL
LIN {X 0,Y 259.727,Z 756.139,A -85,B 0,C 180,E1 -18346.93,E2 -18346.93} C_VEL
LIN {X 0,Y 261.63,Z 753.292,A -85,B 0,C 180,E1 -18349.944,E2 -18349.944} C_VEL
LIN {X 0,Y 263.554,Z 749.714,A -85,B 0,C 180,E1 -18352.338,E2 -18352.338} C_VEL
LIN {X 0,Y 265.747,Z 744.938,A -85,B 0,C 180,E1 -18354.689,E2 -18354.689} C_VEL
LIN {X 0,Y 268.256,Z 738.771,A -85,B 0,C 180,E1 -18356.996,E2 -18356.996} C_VEL
LIN {X 0,Y 271.046,Z 731.014,A -85,B 0,C 180,E1 -18359.257,E2 -18359.257} C_VEL
LIN {X 0,Y 273.511,Z 723.058,A -85,B 0,C 180,E1 -18361.104,E2 -18361.104} C_VEL
LIN {X 0,Y 276.104,Z 713.398,A -85,B 0,C 180,E1 -18362.918,E2 -18362.918} C_VEL
LIN {X 0,Y 278.656,Z 702.612,A -85,B 0,C 180,E1 -18364.52,E2 -18364.52} C_VEL
LIN {X 0,Y 280.824,Z 690.603,A -85,B 0,C 180,E1 -18365.925,E2 -18365.925} C_VEL
LIN {X 0,Y 282.628,Z 677.919,A -85,B 0,C 180,E1 -18367.052,E2 -18367.052} C_VEL
LIN {X 0,Y 283.734,Z 664.94,A -85,B 0,C 180,E1 -18367.929,E2 -18367.929} C_VEL
LIN {X 0,Y 284.994,Z 643.058,A -85,B 0,C 180,E1 -18368.923,E2 -18368.923} C_VEL
LIN {X 0,Y 287.155,Z 614.629,A -85,B 0,C 180,E1 -18370.015,E2 -18370.015} C_VEL
LIN {X 0,Y 282.858,Z 606.037,A -85,B 0,C 180,E1 -18371.578,E2 -18371.578} C_VEL
LIN {X 0,Y 278.938,Z 599.701,A -85,B 0,C 180,E1 -18373.061,E2 -18373.061} C_VEL
LIN {X 0,Y 276.953,Z 596.599,A -85,B 0,C 180,E1 -18373.889,E2 -18373.889} C_VEL
LIN {X 0,Y 274.664,Z 593.169,A -85,B 0,C 180,E1 -18374.878,E2 -18374.878} C_VEL
LIN {X 0,Y 272,Z 589.213,A -85,B 0,C 180,E1 -18376.138,E2 -18376.138} C_VEL
LIN {X 0,Y 269.546,Z 585.701,A -85,B 0,C 180,E1 -18377.381,E2 -18377.381} C_VEL
LIN {X 0,Y 266.268,Z 581.856,A -85,B 0,C 180,E1 -18379.215,E2 -18379.215} C_VEL
LIN {X 0,Y 265.323,Z 579.947,A -85,B 0,C 180,E1 -18379.877,E2 -18379.877} C_VEL
LIN {X 0,Y 262.488,Z 577.584,A -85,B 0,C 180,E1 -18381.756,E2 -18381.756} C_VEL
LIN {X 0,Y 261.801,Z 576.842,A -85,B 0,C 180,E1 -18382.283,E2 -18382.283} C_VEL
LIN {X 0,Y 258.572,Z 574.633,A -85,B 0,C 180,E1 -18385.093,E2 -18385.093} C_VEL
LIN {X 0,Y 258.012,Z 574.014,A -85,B 0,C 180,E1 -18385.992,E2 -18385.992} C_VEL
LIN {X 0,Y 258.413,Z 574.844,A -85,B 0,C 180,E1 -18389.511,E2 -18389.511} C_VEL
LIN {X 0,Y 259.558,Z 577.797,A -85,B 0,C 180,E1 -18394.654,E2 -18394.654} C_VEL
LIN {X 0,Y 260.835,Z 581.577,A -85,B 0,C 180,E1 -18398.616,E2 -18398.616} C_VEL
LIN {X 0,Y 262.339,Z 585.869,A -85,B 0,C 180,E1 -18402.047,E2 -18402.047} C_VEL
LIN {X 0,Y 263.733,Z 590.298,A -85,B 0,C 180,E1 -18404.925,E2 -18404.925} C_VEL
LIN {X 0,Y 264.571,Z 593.249,A -85,B 0,C 180,E1 -18406.525,E2 -18406.525} C_VEL
LIN {X 0,Y 269.737,Z 603.038,A -85,B 0,C 180,E1 -18409.566,E2 -18409.566} C_VEL
LIN {X 0,Y 273.617,Z 611.053,A -85,B 0,C 180,E1 -18411.508,E2 -18411.508} C_VEL
LIN {X 0,Y 276.773,Z 618.186,A -85,B 0,C 180,E1 -18412.944,E2 -18412.944} C_VEL
LIN {X 0,Y 278.5,Z 622.5,A -85,B 0,C 180,E1 -18413.708,E2 -18413.708} C_VEL
LIN {X 0,Y 280.504,Z 638.944,A -85,B 0,C 180,E1 -18415.219,E2 -18415.219} C_VEL
LIN {X 0,Y 281.966,Z 656.952,A -85,B 0,C 180,E1 -18416.6,E2 -18416.6} C_VEL
LIN {X 0,Y 282.673,Z 675.769,A -85,B 0,C 180,E1 -18417.762,E2 -18417.762} C_VEL
LIN {X 0,Y 282.541,Z 688.249,A -85,B 0,C 180,E1 -18418.376,E2 -18418.376} C_VEL
LIN {X 0,Y 280.043,Z 717.442,A -85,B 0,C 180,E1 -18419.455,E2 -18419.455} C_VEL
LIN {X 0,Y 278.157,Z 730.709,A -85,B 0,C 180,E1 -18420.172,E2 -18420.172} C_VEL
LIN {X 0,Y 275.422,Z 744.697,A -85,B 0,C 180,E1 -18421.21,E2 -18421.21} C_VEL
LIN {X 0,Y 272.609,Z 756.498,A -85,B 0,C 180,E1 -18422.353,E2 -18422.353} C_VEL
LIN {X 0,Y 269.273,Z 768.606,A -85,B 0,C 180,E1 -18423.87,E2 -18423.87} C_VEL
LIN {X 0,Y 268.701,Z 770.435,A -85,B 0,C 180,E1 -18424.123,E2 -18424.123} C_VEL
LIN {X 0,Y 267.169,Z 782.617,A -85,B 0,C 180,E1 -18425.111,E2 -18425.111} C_VEL
LIN {X 0,Y 265.354,Z 794.361,A -85,B 0,C 180,E1 -18426.387,E2 -18426.387} C_VEL
LIN {X 0,Y 263.21,Z 806.018,A -85,B 0,C 180,E1 -18428.051,E2 -18428.051} C_VEL
LIN {X 0,Y 261.111,Z 816.37,A -85,B 0,C 180,E1 -18429.932,E2 -18429.932} C_VEL
LIN {X 0,Y 259.382,Z 824.958,A -85,B 0,C 180,E1 -18431.906,E2 -18431.906} C_VEL
LIN {X 0,Y 257.639,Z 832.904,A -85,B 0,C 180,E1 -18434.172,E2 -18434.172} C_VEL
LIN {X 0,Y 256.154,Z 839.462,A -85,B 0,C 180,E1 -18436.515,E2 -18436.515} C_VEL
LIN {X 0,Y 255.164,Z 844.676,A -85,B 0,C 180,E1 -18438.885,E2 -18438.885} C_VEL
LIN {X 0,Y 254.514,Z 848.709,A -85,B 0,C 180,E1 -18441.266,E2 -18441.266} C_VEL
LIN {X 0,Y 254.161,Z 851.682,A -85,B 0,C 180,E1 -18443.651,E2 -18443.651} C_VEL
LIN {X 0,Y 254.064,Z 853.108,A -85,B 0,C 180,E1 -18445.241,E2 -18445.241} C_VEL
LIN {X 0,Y 254.081,Z 854.116,A -85,B 0,C 180,E1 -18446.83,E2 -18446.83} C_VEL
LIN {X 0,Y 254.12,Z 854.733,A -85,B 0,C 180,E1 -18448.417,E2 -18448.417} C_VEL
LIN {X 0,Y 254.144,Z 854.95,A -85,B 0,C 180,E1 -18450.001,E2 -18450.001} C_VEL
LIN {X 0,Y 254.111,Z 854.722,A -85,B 0,C 180,E1 -18451.586,E2 -18451.586} C_VEL
LIN {X 0,Y 254.059,Z 854.099,A -85,B 0,C 180,E1 -18453.173,E2 -18453.173} C_VEL
LIN {X 0,Y 254.135,Z 852.549,A -85,B 0,C 180,E1 -18455.395,E2 -18455.395} C_VEL
LIN {X 0,Y 254.372,Z 849.745,A -85,B 0,C 180,E1 -18457.942,E2 -18457.942} C_VEL
LIN {X 0,Y 254.912,Z 846.062,A -85,B 0,C 180,E1 -18460.325,E2 -18460.325} C_VEL
LIN {X 0,Y 255.716,Z 841.242,A -85,B 0,C 180,E1 -18462.702,E2 -18462.702} C_VEL
LIN {X 0,Y 257.054,Z 835.149,A -85,B 0,C 180,E1 -18465.055,E2 -18465.055} C_VEL
LIN {X 0,Y 258.739,Z 827.562,A -85,B 0,C 180,E1 -18467.386,E2 -18467.386} C_VEL
LIN {X 0,Y 260.354,Z 819.771,A -85,B 0,C 180,E1 -18469.311,E2 -18469.311} C_VEL
LIN {X 0,Y 262.258,Z 810.242,A -85,B 0,C 180,E1 -18471.21,E2 -18471.21} C_VEL
LIN {X 0,Y 264.354,Z 799.668,A -85,B 0,C 180,E1 -18472.882,E2 -18472.882} C_VEL
LIN {X 0,Y 266.153,Z 789.431,A -85,B 0,C 180,E1 -18474.161,E2 -18474.161} C_VEL
LIN {X 0,Y 267.831,Z 777.149,A -85,B 0,C 180,E1 -18475.345,E2 -18475.345} C_VEL
LIN {X 0,Y 269.285,Z 764.271,A -85,B 0,C 180,E1 -18476.236,E2 -18476.236} C_VEL
LIN {X 0,Y 270.335,Z 751.532,A -85,B 0,C 180,E1 -18476.802,E2 -18476.802} C_VEL
LIN {X 0,Y 272.338,Z 684.769,A -85,B 0,C 180,E1 -18478.562,E2 -18478.562} C_VEL
LIN {X 0,Y 269.559,Z 656.331,A -85,B 0,C 180,E1 -18479.73,E2 -18479.73} C_VEL
LIN {X 0,Y 266.68,Z 634.121,A -85,B 0,C 180,E1 -18480.808,E2 -18480.808} C_VEL
LIN {X 0,Y 265.773,Z 606.515,A -85,B 0,C 180,E1 -18483.733,E2 -18483.733} C_VEL
LIN {X 0,Y 265.334,Z 603.06,A -85,B 0,C 180,E1 -18484.133,E2 -18484.133} C_VEL
LIN {X 0,Y 261.63,Z 590.952,A -85,B 0,C 180,E1 -18485.982,E2 -18485.982} C_VEL
LIN {X 0,Y 259.524,Z 584.274,A -85,B 0,C 180,E1 -18487.063,E2 -18487.063} C_VEL
LIN {X 0,Y 256.857,Z 571.95,A -85,B 0,C 180,E1 -18491.048,E2 -18491.048} C_VEL
LIN {X 0,Y 256.095,Z 568.586,A -85,B 0,C 180,E1 -18492.187,E2 -18492.187} C_VEL
LIN {X 0,Y 256.068,Z 568.586,A -85,B 0,C 180,E1 -18496.674,E2 -18496.674} C_VEL
LIN {X 0,Y 256.074,Z 568.589,A -85,B 0,C 180,E1 -18500.858,E2 -18500.858} C_VEL
LIN {X 0,Y 256.132,Z 568.563,A -85,B 0,C 180,E1 -18502.868,E2 -18502.868} C_VEL
LIN {X 0,Y 256.07,Z 568.586,A -85,B 0,C 180,E1 -18506.708,E2 -18506.708} C_VEL
LIN {X 0,Y 256.116,Z 568.57,A -85,B 0,C 180,E1 -18510.401,E2 -18510.401} C_VEL
LIN {X 0,Y 256.173,Z 568.551,A -85,B 0,C 180,E1 -18514.87,E2 -18514.87} C_VEL
LIN {X 0,Y 256.165,Z 568.577,A -85,B 0,C 180,E1 -18519.105,E2 -18519.105} C_VEL
LIN {X 0,Y 256.282,Z 568.547,A -85,B 0,C 180,E1 -18524.084,E2 -18524.084} C_VEL
LIN {X 0,Y 256.296,Z 568.549,A -85,B 0,C 180,E1 -18527.328,E2 -18527.328} C_VEL
LIN {X 0,Y 256.518,Z 568.525,A -85,B 0,C 180,E1 -18532.126,E2 -18532.126} C_VEL
LIN {X 0,Y 256.499,Z 568.504,A -85,B 0,C 180,E1 -18536.859,E2 -18536.859} C_VEL
LIN {X 0,Y 256.76,Z 568.496,A -85,B 0,C 180,E1 -18540,E2 -18540} C_VEL
LIN {X 0,Y 256.499,Z 568.519,A -85,B 0,C 180,E1 -18543.141,E2 -18543.141} C_VEL
LIN {X 0,Y 256.54,Z 568.525,A -85,B 0,C 180,E1 -18547.873,E2 -18547.873} C_VEL
LIN {X 0,Y 256.312,Z 568.538,A -85,B 0,C 180,E1 -18551.066,E2 -18551.066} C_VEL
LIN {X 0,Y 256.298,Z 568.562,A -85,B 0,C 180,E1 -18555.915,E2 -18555.915} C_VEL
LIN {X 0,Y 256.17,Z 568.563,A -85,B 0,C 180,E1 -18560.895,E2 -18560.895} C_VEL
LIN {X 0,Y 256.191,Z 568.552,A -85,B 0,C 180,E1 -18565.138,E2 -18565.138} C_VEL
LIN {X 0,Y 256.116,Z 568.572,A -85,B 0,C 180,E1 -18569.6,E2 -18569.6} C_VEL
LIN {X 0,Y 256.071,Z 568.591,A -85,B 0,C 180,E1 -18573.293,E2 -18573.293} C_VEL
LIN {X 0,Y 256.128,Z 568.584,A -85,B 0,C 180,E1 -18577.274,E2 -18577.274} C_VEL
LIN {X 0,Y 256.06,Z 568.592,A -85,B 0,C 180,E1 -18581.203,E2 -18581.203} C_VEL
LIN {X 0,Y 256.074,Z 568.657,A -85,B 0,C 180,E1 -18584.41,E2 -18584.41} C_VEL
LIN {X 0,Y 260.703,Z 581.372,A -85,B 0,C 180,E1 -18588.424,E2 -18588.424} C_VEL
LIN {X 0,Y 264.346,Z 593.044,A -85,B 0,C 180,E1 -18591.756,E2 -18591.756} C_VEL
LIN {X 0,Y 266.858,Z 602.756,A -85,B 0,C 180,E1 -18594.334,E2 -18594.334} C_VEL
LIN {X 0,Y 269.425,Z 614.67,A -85,B 0,C 180,E1 -18597.271,E2 -18597.271} C_VEL
LIN {X 0,Y 268.354,Z 625.481,A -85,B 0,C 180,E1 -18599.313,E2 -18599.313} C_VEL
LIN {X 0,Y 268.86,Z 628.99,A -85,B 0,C 180,E1 -18599.544,E2 -18599.544} C_VEL
LIN {X 0,Y 273.007,Z 655.38,A -85,B 0,C 180,E1 -18600.841,E2 -18600.841} C_VEL
LIN {X 0,Y 273.671,Z 661.775,A -85,B 0,C 180,E1 -18601.108,E2 -18601.108} C_VEL
LIN {X 0,Y 271.097,Z 738.528,A -85,B 0,C 180,E1 -18603.123,E2 -18603.123} C_VEL
LIN {X 0,Y 270.142,Z 751.647,A -85,B 0,C 180,E1 -18603.75,E2 -18603.75} C_VEL
LIN {X 0,Y 268.807,Z 764.122,A -85,B 0,C 180,E1 -18604.65,E2 -18604.65} C_VEL
LIN {X 0,Y 267.281,Z 775.326,A -85,B 0,C 180,E1 -18605.741,E2 -18605.741} C_VEL
LIN {X 0,Y 265.293,Z 786.912,A -85,B 0,C 180,E1 -18607.204,E2 -18607.204} C_VEL
LIN {X 0,Y 263.316,Z 797.664,A -85,B 0,C 180,E1 -18608.961,E2 -18608.961} C_VEL
LIN {X 0,Y 261.601,Z 806.58,A -85,B 0,C 180,E1 -18610.785,E2 -18610.785} C_VEL
LIN {X 0,Y 259.816,Z 814.229,A -85,B 0,C 180,E1 -18612.688,E2 -18612.688} C_VEL
LIN {X 0,Y 258.044,Z 821.685,A -85,B 0,C 180,E1 -18615.004,E2 -18615.004} C_VEL
LIN {X 0,Y 256.649,Z 827.67,A -85,B 0,C 180,E1 -18617.344,E2 -18617.344} C_VEL
LIN {X 0,Y 255.579,Z 832.399,A -85,B 0,C 180,E1 -18619.703,E2 -18619.703} C_VEL
LIN {X 0,Y 254.884,Z 836.011,A -85,B 0,C 180,E1 -18622.074,E2 -18622.074} C_VEL
LIN {X 0,Y 254.51,Z 837.999,A -85,B 0,C 180,E1 -18623.775,E2 -18623.775} C_VEL
LIN {X 0,Y 254.165,Z 840.283,A -85,B 0,C 180,E1 -18626.829,E2 -18626.829} C_VEL
